	LOCAL CONST Robtarget Tr_meulage_bavure_P136 :=[[-151.101640625,13.911193359375,23],[0.363113173339064,-0.403939689053268,0.624425765586211,-0.561314541257626],[0,0,0,0],[8.999999E+09,8.999999E+09,8.999999E+09,8.999999E+09,8.999999E+09,8.999999E+09]];
	LOCAL CONST Robtarget Tr_meulage_bavure_P137 :=[[-149.937296875,16.62026953125,23],[0.361366142392558,-0.400488127447699,0.625160151915924,-0.564090910547419],[0,0,0,0],[8.999999E+09,8.999999E+09,8.999999E+09,8.999999E+09,8.999999E+09,8.999999E+09]];
	LOCAL CONST Robtarget Tr_meulage_bavure_P138 :=[[-148.7885625,19.131255859375,23],[0.359765710075978,-0.397152746767946,0.625734149066699,-0.566828990331279],[0,0,0,0],[8.999999E+09,8.999999E+09,8.999999E+09,8.999999E+09,8.999999E+09,8.999999E+09]];
	LOCAL CONST Robtarget Tr_meulage_bavure_P139 :=[[-148.23471875,20.335998046875,23],[0.358570112588793,-0.394222003460565,0.625973297444358,-0.569362729050853],[0,0,0,0],[8.999999E+09,8.999999E+09,8.999999E+09,8.999999E+09,8.999999E+09,8.999999E+09]];
	LOCAL CONST Robtarget Tr_meulage_bavure_P140 :=[[-145.765296875,25.489470703125,23],[0.35796569299165,-0.39191876694484,0.625767359146769,-0.571555294773763],[0,0,0,0],[8.999999E+09,8.999999E+09,8.999999E+09,8.999999E+09,8.999999E+09,8.999999E+09]];
	LOCAL CONST Robtarget Tr_meulage_bavure_P141 :=[[-144.20271875,28.765869140625,23],[0.358018242776586,-0.390330323158982,0.625091784203007,-0.573345827562799],[0,0,0,0],[8.999999E+09,8.999999E+09,8.999999E+09,8.999999E+09,8.999999E+09,8.999999E+09]];
	LOCAL CONST Robtarget Tr_meulage_bavure_P142 :=[[-143.79815625,29.5517578125,23],[0.358645064931337,-0.3893852969019,0.624023000869993,-0.57475916899361],[0,0,0,0],[8.999999E+09,8.999999E+09,8.999999E+09,8.999999E+09,8.999999E+09,8.999999E+09]];
	LOCAL CONST Robtarget Tr_meulage_bavure_P143 :=[[-142.6278125,32.183806640625,23],[0.359633831929679,-0.388864753981572,0.622717813839782,-0.575908182238306],[0,0,0,0],[8.999999E+09,8.999999E+09,8.999999E+09,8.999999E+09,8.999999E+09,8.999999E+09]];
	LOCAL CONST Robtarget Tr_meulage_bavure_P144 :=[[-141.08978125,35.4830625,23],[0.360692368664617,-0.388472413246163,0.621385243175179,-0.576949372907133],[0,0,0,0],[8.999999E+09,8.999999E+09,8.999999E+09,8.999999E+09,8.999999E+09,8.999999E+09]];
	LOCAL CONST Robtarget Tr_meulage_bavure_P145 :=[[-140.90496875,35.88940625,23],[0.36152355469278,-0.387927178958205,0.620241455843297,-0.578025743095594],[0,0,0,0],[8.999999E+09,8.999999E+09,8.999999E+09,8.999999E+09,8.999999E+09,8.999999E+09]];
	LOCAL CONST Robtarget Tr_meulage_bavure_P146 :=[[-140.313296875,37.1786796875,23],[0.361932466131916,-0.387033912571134,0.619420641915412,-0.579247536765284],[0,0,0,0],[8.999999E+09,8.999999E+09,8.999999E+09,8.999999E+09,8.999999E+09,8.999999E+09]];
	LOCAL CONST Robtarget Tr_meulage_bavure_P147 :=[[-139.0531875,39.5576171875,23],[0.361853147250191,-0.385747951920083,0.618973239019357,-0.580631506889248],[0,0,0,0],[8.999999E+09,8.999999E+09,8.999999E+09,8.999999E+09,8.999999E+09,8.999999E+09]];
	LOCAL CONST Robtarget Tr_meulage_bavure_P148 :=[[-138.05065625,41.53494140625,23],[0.361341124651924,-0.384146531890856,0.618865172241677,-0.582125357854981],[0,0,0,0],[8.999999E+09,8.999999E+09,8.999999E+09,8.999999E+09,8.999999E+09,8.999999E+09]];
	LOCAL CONST Robtarget Tr_meulage_bavure_P149 :=[[-136.388,44.438078125,23],[0.360507751556033,-0.382372963113046,0.619030246412353,-0.583632274788522],[0,0,0,0],[8.999999E+09,8.999999E+09,8.999999E+09,8.999999E+09,8.999999E+09,8.999999E+09]];
	LOCAL CONST Robtarget Tr_meulage_bavure_P150 :=[[-135.13509375,47.07137890625,23],[0.359446609197695,-0.380538333002904,0.619411292399243,-0.585079792079636],[0,0,0,0],[8.999999E+09,8.999999E+09,8.999999E+09,8.999999E+09,8.999999E+09,8.999999E+09]];
	LOCAL CONST Robtarget Tr_meulage_bavure_P151 :=[[-133.055,51.51773046875,23],[0.358189967630797,-0.378660333676248,0.61998050741984,-0.586464380170082],[0,0,0,0],[8.999999E+09,8.999999E+09,8.999999E+09,8.999999E+09,8.999999E+09,8.999999E+09]];
	LOCAL CONST Robtarget Tr_meulage_bavure_P152 :=[[-132.991484375,51.62383984375,23],[0.356688173346148,-0.376690925174669,0.620772461958371,-0.587808680065362],[0,0,0,0],[8.999999E+09,8.999999E+09,8.999999E+09,8.999999E+09,8.999999E+09,8.999999E+09]];
	LOCAL CONST Robtarget Tr_meulage_bavure_P153 :=[[-132.88184375,51.8467109375,23],[0.354871689037836,-0.374562381729461,0.621834258118938,-0.589144517026389],[0,0,0,0],[8.999999E+09,8.999999E+09,8.999999E+09,8.999999E+09,8.999999E+09,8.999999E+09]];
	LOCAL CONST Robtarget Tr_meulage_bavure_P154 :=[[-132.33325,52.87548828125,23],[0.352738855187171,-0.372246378330528,0.623153787667112,-0.590497494302203],[0,0,0,0],[8.999999E+09,8.999999E+09,8.999999E+09,8.999999E+09,8.999999E+09,8.999999E+09]];
	LOCAL CONST Robtarget Tr_meulage_bavure_P155 :=[[-129.2417578125,58.37216015625,23],[0.350372889166439,-0.36982520954016,0.624675359558615,-0.591818255958748],[0,0,0,0],[8.999999E+09,8.999999E+09,8.999999E+09,8.999999E+09,8.999999E+09,8.999999E+09]];
	LOCAL CONST Robtarget Tr_meulage_bavure_P156 :=[[-128.5902734375,59.6175234375,23],[0.347952755656077,-0.367462162625027,0.626275780687696,-0.593025366569001],[0,0,0,0],[8.999999E+09,8.999999E+09,8.999999E+09,8.999999E+09,8.999999E+09,8.999999E+09]];
	LOCAL CONST Robtarget Tr_meulage_bavure_P157 :=[[-128.01315625,60.49066015625,23],[0.345666878551163,-0.365345597032472,0.627836321567684,-0.594018987173004],[0,0,0,0],[8.999999E+09,8.999999E+09,8.999999E+09,8.999999E+09,8.999999E+09,8.999999E+09]];
	LOCAL CONST Robtarget Tr_meulage_bavure_P158 :=[[-126.7691640625,62.76187109375,23],[0.343644652538738,-0.363593971431505,0.629272863290692,-0.594746534454914],[0,0,0,0],[8.999999E+09,8.999999E+09,8.999999E+09,8.999999E+09,8.999999E+09,8.999999E+09]];
	LOCAL CONST Robtarget Tr_meulage_bavure_P159 :=[[-125.6860078125,64.59457421875,23],[0.341903861092431,-0.362214737571814,0.630573008552044,-0.595214175353287],[0,0,0,0],[8.999999E+09,8.999999E+09,8.999999E+09,8.999999E+09,8.999999E+09,8.999999E+09]];
	LOCAL CONST Robtarget Tr_meulage_bavure_P160 :=[[-124.4326484375,66.62625,23],[0.340355790714089,-0.361121197706101,0.63179741148611,-0.595467419036633],[0,0,0,0],[8.999999E+09,8.999999E+09,8.999999E+09,8.999999E+09,8.999999E+09,8.999999E+09]];
	LOCAL CONST Robtarget Tr_meulage_bavure_P161 :=[[-123.00375,69.2471953125,23],[0.338884891304971,-0.360167100503058,0.633005414582959,-0.59560123847176],[0,0,0,0],[8.999999E+09,8.999999E+09,8.999999E+09,8.999999E+09,8.999999E+09,8.999999E+09]];
	LOCAL CONST Robtarget Tr_meulage_bavure_P162 :=[[-122.3022734375,70.33459375,23],[0.33739329406918,-0.359234517684621,0.634249603211876,-0.595687642348424],[0,0,0,0],[8.999999E+09,8.999999E+09,8.999999E+09,8.999999E+09,8.999999E+09,8.999999E+09]];
	LOCAL CONST Robtarget Tr_meulage_bavure_P163 :=[[-121.89965625,71.103359375,23],[0.335824905230539,-0.358297647661144,0.635582135777234,-0.595717867272956],[0,0,0,0],[8.999999E+09,8.999999E+09,8.999999E+09,8.999999E+09,8.999999E+09,8.999999E+09]];
	LOCAL CONST Robtarget Tr_meulage_bavure_P164 :=[[-121.4621875,71.8283046875,23],[0.334205475423421,-0.35736441895173,0.636977751618542,-0.595698511167591],[0,0,0,0],[8.999999E+09,8.999999E+09,8.999999E+09,8.999999E+09,8.999999E+09,8.999999E+09]];
	LOCAL CONST Robtarget Tr_meulage_bavure_P165 :=[[-116.748078125,79.6233828125,23],[0.332558951177178,-0.356471847846565,0.638428689604975,-0.595601522810398],[0,0,0,0],[8.999999E+09,8.999999E+09,8.999999E+09,8.999999E+09,8.999999E+09,8.999999E+09]];
	LOCAL CONST Robtarget Tr_meulage_bavure_P166 :=[[-116.44934375,80.07165625,23],[0.33089213683516,-0.355635671324102,0.639935992215293,-0.595412116882034],[0,0,0,0],[8.999999E+09,8.999999E+09,8.999999E+09,8.999999E+09,8.999999E+09,8.999999E+09]];
	LOCAL CONST Robtarget Tr_meulage_bavure_P167 :=[[-115.361484375,81.8792109375,23],[0.329186352606248,-0.354835404169223,0.641511190202099,-0.595139961732823],[0,0,0,0],[8.999999E+09,8.999999E+09,8.999999E+09,8.999999E+09,8.999999E+09,8.999999E+09]];
	LOCAL CONST Robtarget Tr_meulage_bavure_P168 :=[[-112.9508046875,85.6936953125,23],[0.32739769262739,-0.354043304067062,0.64319165616197,-0.594784484625449],[0,0,0,0],[8.999999E+09,8.999999E+09,8.999999E+09,8.999999E+09,8.999999E+09,8.999999E+09]];
	LOCAL CONST Robtarget Tr_meulage_bavure_P169 :=[[-110.774625,89.2081015625,23],[0.325512172612704,-0.353248750896646,0.644988949272338,-0.59434535481274],[0,0,0,0],[8.999999E+09,8.999999E+09,8.999999E+09,8.999999E+09,8.999999E+09,8.999999E+09]];
	LOCAL CONST Robtarget Tr_meulage_bavure_P170 :=[[-110.4715,89.681578125,23],[0.323541727027112,-0.352470758041441,0.646900127086222,-0.593805810997026],[0,0,0,0],[8.999999E+09,8.999999E+09,8.999999E+09,8.999999E+09,8.999999E+09,8.999999E+09]];
	LOCAL CONST Robtarget Tr_meulage_bavure_P171 :=[[-110.3179609375,89.93865625,23],[0.321490986582534,-0.351726089874816,0.648929676846336,-0.593146337555642],[0,0,0,0],[8.999999E+09,8.999999E+09,8.999999E+09,8.999999E+09,8.999999E+09,8.999999E+09]];
	LOCAL CONST Robtarget Tr_meulage_bavure_P172 :=[[-108.4508984375,92.7417578125,23],[0.319339852371983,-0.350964788325318,0.6510751687394,-0.592407714917494],[0,0,0,0],[8.999999E+09,8.999999E+09,8.999999E+09,8.999999E+09,8.999999E+09,8.999999E+09]];
	LOCAL CONST Robtarget Tr_meulage_bavure_P173 :=[[-107.08996875,94.77328125,23],[0.316996000347298,-0.350097784864441,0.653399226164253,-0.59162025662141],[0,0,0,0],[8.999999E+09,8.999999E+09,8.999999E+09,8.999999E+09,8.999999E+09,8.999999E+09]];
	LOCAL CONST Robtarget Tr_meulage_bavure_P174 :=[[-105.537234375,96.8504296875,23],[0.314366480436105,-0.349013203905433,0.655953733645348,-0.590836863097259],[0,0,0,0],[8.999999E+09,8.999999E+09,8.999999E+09,8.999999E+09,8.999999E+09,8.999999E+09]];
	LOCAL CONST Robtarget Tr_meulage_bavure_P175 :=[[-104.5172421875,98.662203125,23],[0.311427948746812,-0.347654360016432,0.658738048574652,-0.590095976991012],[0,0,0,0],[8.999999E+09,8.999999E+09,8.999999E+09,8.999999E+09,8.999999E+09,8.999999E+09]];
	LOCAL CONST Robtarget Tr_meulage_bavure_P176 :=[[-104.1592421875,99.2328828125,23],[0.308276601042876,-0.346110430708768,0.661687715989301,-0.589357678759601],[0,0,0,0],[8.999999E+09,8.999999E+09,8.999999E+09,8.999999E+09,8.999999E+09,8.999999E+09]];
	LOCAL CONST Robtarget Tr_meulage_bavure_P177 :=[[-103.0036953125,100.7189609375,23],[0.305135247230992,-0.344604748309039,0.664658435505481,-0.588531403114186],[0,0,0,0],[8.999999E+09,8.999999E+09,8.999999E+09,8.999999E+09,8.999999E+09,8.999999E+09]];
	LOCAL CONST Robtarget Tr_meulage_bavure_P178 :=[[-102.00121875,102.1814609375,23],[0.302287241198627,-0.343432763280974,0.66747032690831,-0.587502956256929],[0,0,0,0],[8.999999E+09,8.999999E+09,8.999999E+09,8.999999E+09,8.999999E+09,8.999999E+09]];
	LOCAL CONST Robtarget Tr_meulage_bavure_P179 :=[[-97.7013515625,108.074984375,23],[0.299987070179315,-0.342864199056344,0.669960522310556,-0.586178127599494],[0,0,0,0],[8.999999E+09,8.999999E+09,8.999999E+09,8.999999E+09,8.999999E+09,8.999999E+09]];
	LOCAL CONST Robtarget Tr_meulage_bavure_P180 :=[[-97.20065625,108.7268046875,23],[0.298390218171339,-0.343046324630686,0.672013629572218,-0.584534155140837],[0,0,0,0],[8.999999E+09,8.999999E+09,8.999999E+09,8.999999E+09,8.999999E+09,8.999999E+09]];
	LOCAL CONST Robtarget Tr_meulage_bavure_P181 :=[[-96.925140625,109.1156953125,23],[0.297488777694042,-0.343974793916163,0.673625579809489,-0.582589346386258],[0,0,0,0],[8.999999E+09,8.999999E+09,8.999999E+09,8.999999E+09,8.999999E+09,8.999999E+09]];
	LOCAL CONST Robtarget Tr_meulage_bavure_P182 :=[[-96.654234375,109.4932890625,23],[0.297146717753407,-0.345460993457581,0.674847244361684,-0.58046681809137],[0,0,0,0],[8.999999E+09,8.999999E+09,8.999999E+09,8.999999E+09,8.999999E+09,8.999999E+09]];
	LOCAL CONST Robtarget Tr_meulage_bavure_P183 :=[[-93.7308671875,113.3792734375,23],[0.297098761957459,-0.347164074281642,0.675810702966835,-0.578350520815005],[0,0,0,0],[8.999999E+09,8.999999E+09,8.999999E+09,8.999999E+09,8.999999E+09,8.999999E+09]];
	LOCAL CONST Robtarget Tr_meulage_bavure_P184 :=[[-90.1459375,118.35940625,23],[0.296995083840805,-0.348662276006968,0.6767185983147,-0.576437746993568],[0,0,0,0],[8.999999E+09,8.999999E+09,8.999999E+09,8.999999E+09,8.999999E+09,8.999999E+09]];
	LOCAL CONST Robtarget Tr_meulage_bavure_P185 :=[[-89.706484375,118.935421875,23],[0.296477938104876,-0.34949723785255,0.677774921241467,-0.574955362690569],[0,0,0,0],[8.999999E+09,8.999999E+09,8.999999E+09,8.999999E+09,8.999999E+09,8.999999E+09]];
	LOCAL CONST Robtarget Tr_meulage_bavure_P186 :=[[-89.5105,119.176546875,23],[0.295232063451212,-0.349274248056214,0.679170511051546,-0.574084440890961],[0,0,0,0],[8.999999E+09,8.999999E+09,8.999999E+09,8.999999E+09,8.999999E+09,8.999999E+09]];
	LOCAL CONST Robtarget Tr_meulage_bavure_P187 :=[[-89.0611875,119.83196875,23],[0.293080552541801,-0.347759738084034,0.681007104196331,-0.573930551829787],[0,0,0,0],[8.999999E+09,8.999999E+09,8.999999E+09,8.999999E+09,8.999999E+09,8.999999E+09]];
	LOCAL CONST Robtarget Tr_meulage_bavure_P188 :=[[-87.366484375,122.046390625,23],[0.290040566264844,-0.344934373310814,0.683249092361541,-0.574514948296887],[0,0,0,0],[8.999999E+09,8.999999E+09,8.999999E+09,8.999999E+09,8.999999E+09,8.999999E+09]];
	LOCAL CONST Robtarget Tr_meulage_bavure_P189 :=[[-85.4241328125,124.5614921875,23],[0.286302590251918,-0.341056323606131,0.685782309095291,-0.575685708937823],[0,0,0,0],[8.999999E+09,8.999999E+09,8.999999E+09,8.999999E+09,8.999999E+09,8.999999E+09]];
	LOCAL CONST Robtarget Tr_meulage_bavure_P190 :=[[-82.9652109375,127.53896875,23],[0.282238780633603,-0.336559090185623,0.688360590316553,-0.577259861084182],[0,0,0,0],[8.999999E+09,8.999999E+09,8.999999E+09,8.999999E+09,8.999999E+09,8.999999E+09]];
	LOCAL CONST Robtarget Tr_meulage_bavure_P191 :=[[-80.8466171875,130.312015625,23],[0.278274994959359,-0.331954569840343,0.690722014669287,-0.579027019398648],[0,0,0,0],[8.999999E+09,8.999999E+09,8.999999E+09,8.999999E+09,8.999999E+09,8.999999E+09]];
	LOCAL CONST Robtarget Tr_meulage_bavure_P192 :=[[-80.806546875,130.3608671875,23],[0.274742616549122,-0.327682985270072,0.692696966908732,-0.580785044445601],[0,0,0,0],[8.999999E+09,8.999999E+09,8.999999E+09,8.999999E+09,8.999999E+09,8.999999E+09]];
	LOCAL CONST Robtarget Tr_meulage_bavure_P193 :=[[-80.775234375,130.400515625,23],[0.271819685652551,-0.323980055433208,0.694203028496095,-0.582437239022449],[0,0,0,0],[8.999999E+09,8.999999E+09,8.999999E+09,8.999999E+09,8.999999E+09,8.999999E+09]];
	LOCAL CONST Robtarget Tr_meulage_bavure_P194 :=[[-80.66,130.534453125,23],[0.269492995590509,-0.320855422562745,0.69527098544135,-0.583972242442352],[0,0,0,0],[8.999999E+09,8.999999E+09,8.999999E+09,8.999999E+09,8.999999E+09,8.999999E+09]];
	LOCAL CONST Robtarget Tr_meulage_bavure_P195 :=[[-75.0816015625,136.849671875,23],[0.267608889300657,-0.318155220259668,0.696010587349302,-0.585433173373759],[0,0,0,0],[8.999999E+09,8.999999E+09,8.999999E+09,8.999999E+09,8.999999E+09,8.999999E+09]];
	LOCAL CONST Robtarget Tr_meulage_bavure_P196 :=[[-73.9031640625,138.106265625,23],[0.265971457519477,-0.315679629512676,0.696553803832876,-0.586871667114418],[0,0,0,0],[8.999999E+09,8.999999E+09,8.999999E+09,8.999999E+09,8.999999E+09,8.999999E+09]];
	LOCAL CONST Robtarget Tr_meulage_bavure_P197 :=[[-70.499453125,142.30071875,23],[0.264424748051487,-0.313302265360263,0.697024796870706,-0.588283669402258],[0,0,0,0],[8.999999E+09,8.999999E+09,8.999999E+09,8.999999E+09,8.999999E+09,8.999999E+09]];
	LOCAL CONST Robtarget Tr_meulage_bavure_P198 :=[[-69.435421875,143.518640625,23],[0.262940352786829,-0.311003055889999,0.69744901940964,-0.589664595705009],[0,0,0,0],[8.999999E+09,8.999999E+09,8.999999E+09,8.999999E+09,8.999999E+09,8.999999E+09]];
	LOCAL CONST Robtarget Tr_meulage_bavure_P199 :=[[-67.65221875,145.57946875,23],[0.26158305272051,-0.308882913750533,0.697810610604228,-0.590953470123117],[0,0,0,0],[8.999999E+09,8.999999E+09,8.999999E+09,8.999999E+09,8.999999E+09,8.999999E+09]];
	LOCAL CONST Robtarget Tr_meulage_bavure_P200 :=[[-63.85848828125,149.82321875,23],[0.260452446063248,-0.307115703409703,0.698100327852684,-0.592030742707512],[0,0,0,0],[8.999999E+09,8.999999E+09,8.999999E+09,8.999999E+09,8.999999E+09,8.999999E+09]];
	LOCAL CONST Robtarget Tr_meulage_bavure_P201 :=[[-62.9795546875,150.73965625,23],[0.259650622045114,-0.305842532734676,0.698285923040029,-0.592822628891778],[0,0,0,0],[8.999999E+09,8.999999E+09,8.999999E+09,8.999999E+09,8.999999E+09,8.999999E+09]];
	LOCAL CONST Robtarget Tr_meulage_bavure_P202 :=[[-60.04244921875,154.120734375,23],[0.25923435549752,-0.305149200328328,0.698357387354537,-0.593277737654222],[0,0,0,0],[8.999999E+09,8.999999E+09,8.999999E+09,8.999999E+09,8.999999E+09,8.999999E+09]];
	LOCAL CONST Robtarget Tr_meulage_bavure_P203 :=[[-58.3733515625,155.91925,23],[0.259193420326712,-0.305039549462365,0.698335046608728,-0.593378299907507],[0,0,0,0],[8.999999E+09,8.999999E+09,8.999999E+09,8.999999E+09,8.999999E+09,8.999999E+09]];
	LOCAL CONST Robtarget Tr_meulage_bavure_P204 :=[[-57.8063046875,156.5224375,23],[0.259457229635472,-0.305442867370749,0.698264748264398,-0.593138215000077],[0,0,0,0],[8.999999E+09,8.999999E+09,8.999999E+09,8.999999E+09,8.999999E+09,8.999999E+09]];
	LOCAL CONST Robtarget Tr_meulage_bavure_P205 :=[[-53.8414921875,160.451046875,23],[0.259910866387483,-0.306232150271341,0.698209736878708,-0.592597143936473],[0,0,0,0],[8.999999E+09,8.999999E+09,8.999999E+09,8.999999E+09,8.999999E+09,8.999999E+09]];
	LOCAL CONST Robtarget Tr_meulage_bavure_P206 :=[[-51.208921875,163.25109375,23],[0.260395135511095,-0.307211321910998,0.698243437299184,-0.591837544737132],[0,0,0,0],[8.999999E+09,8.999999E+09,8.999999E+09,8.999999E+09,8.999999E+09,8.999999E+09]];
	LOCAL CONST Robtarget Tr_meulage_bavure_P207 :=[[-48.69293359375,165.973234375,23],[0.260708052450437,-0.308133124993847,0.698462495975598,-0.590961445768304],[0,0,0,0],[8.999999E+09,8.999999E+09,8.999999E+09,8.999999E+09,8.999999E+09,8.999999E+09]];
	LOCAL CONST Robtarget Tr_meulage_bavure_P208 :=[[-47.96395703125,166.6900625,23],[0.260627562818114,-0.308725558365438,0.698976562907696,-0.590079289263047],[0,0,0,0],[8.999999E+09,8.999999E+09,8.999999E+09,8.999999E+09,8.999999E+09,8.999999E+09]];
	LOCAL CONST Robtarget Tr_meulage_bavure_P209 :=[[-47.6884453125,166.9998125,23],[0.259952138246991,-0.308717659214279,0.699872182769465,-0.589319285697981],[0,0,0,0],[8.999999E+09,8.999999E+09,8.999999E+09,8.999999E+09,8.999999E+09,8.999999E+09]];
	LOCAL CONST Robtarget Tr_meulage_bavure_P210 :=[[-47.49398828125,167.2056875,23],[0.258524685420064,-0.307880894401815,0.70120753717733,-0.588797360470051],[0,0,0,0],[8.999999E+09,8.999999E+09,8.999999E+09,8.999999E+09,8.999999E+09,8.999999E+09]];
	LOCAL CONST Robtarget Tr_meulage_bavure_P211 :=[[-46.68640234375,168.037875,23],[0.256255031366667,-0.306077422500699,0.703012135818707,-0.588577868447512],[0,0,0,0],[8.999999E+09,8.999999E+09,8.999999E+09,8.999999E+09,8.999999E+09,8.999999E+09]];
	LOCAL CONST Robtarget Tr_meulage_bavure_P212 :=[[-42.5556953125,172.1044375,23],[0.253174527212128,-0.303299309659537,0.705237754876775,-0.588686586077285],[0,0,0,0],[8.999999E+09,8.999999E+09,8.999999E+09,8.999999E+09,8.999999E+09,8.999999E+09]];
	LOCAL CONST Robtarget Tr_meulage_bavure_P213 :=[[-41.41424609375,173.362859375,23],[0.249437788419242,-0.299696304442926,0.707774725152081,-0.589082212639006],[0,0,0,0],[8.999999E+09,8.999999E+09,8.999999E+09,8.999999E+09,8.999999E+09,8.999999E+09]];
	LOCAL CONST Robtarget Tr_meulage_bavure_P214 :=[[-39.20593359375,175.651515625,23],[0.245328958803579,-0.29556827111994,0.710440992387538,-0.589683555320082],[0,0,0,0],[8.999999E+09,8.999999E+09,8.999999E+09,8.999999E+09,8.999999E+09,8.999999E+09]];
	LOCAL CONST Robtarget Tr_meulage_bavure_P215 :=[[-34.94815234375,180.011390625,23],[0.241200692788689,-0.291315873340678,0.713035034890375,-0.590371346490408],[0,0,0,0],[8.999999E+09,8.999999E+09,8.999999E+09,8.999999E+09,8.999999E+09,8.999999E+09]];
	LOCAL CONST Robtarget Tr_meulage_bavure_P216 :=[[-34.57086328125,180.35953125,23],[0.237386947714952,-0.287326399661774,0.71537675117121,-0.591038984328196],[0,0,0,0],[8.999999E+09,8.999999E+09,8.999999E+09,8.999999E+09,8.999999E+09,8.999999E+09]];
	LOCAL CONST Robtarget Tr_meulage_bavure_P217 :=[[-33.607484375,181.285671875,23],[0.234098705180864,-0.283854988465174,0.717364032824637,-0.591618953521312],[0,0,0,0],[8.999999E+09,8.999999E+09,8.999999E+09,8.999999E+09,8.999999E+09,8.999999E+09]];
	LOCAL CONST Robtarget Tr_meulage_bavure_P218 :=[[-32.24230859375,182.4925,23],[0.231389418192959,-0.28095490120141,0.718964421329079,-0.592126204032698],[0,0,0,0],[8.999999E+09,8.999999E+09,8.999999E+09,8.999999E+09,8.999999E+09,8.999999E+09]];
	LOCAL CONST Robtarget Tr_meulage_bavure_P219 :=[[-31.390533203125,183.272,23],[0.229147339722196,-0.27850899502818,0.720247483284206,-0.592594126877242],[0,0,0,0],[8.999999E+09,8.999999E+09,8.999999E+09,8.999999E+09,8.999999E+09,8.999999E+09]];
	LOCAL CONST Robtarget Tr_meulage_bavure_P220 :=[[-26.916779296875,187.099859375,23],[0.227187311028143,-0.276294003133417,0.721302168803879,-0.593102630932568],[0,0,0,0],[8.999999E+09,8.999999E+09,8.999999E+09,8.999999E+09,8.999999E+09,8.999999E+09]];
	LOCAL CONST Robtarget Tr_meulage_bavure_P221 :=[[-24.466033203125,189.348875,23],[0.225315180737453,-0.274084145121572,0.722226163804524,-0.593717373030659],[0,0,0,0],[8.999999E+09,8.999999E+09,8.999999E+09,8.999999E+09,8.999999E+09,8.999999E+09]];
	LOCAL CONST Robtarget Tr_meulage_bavure_P222 :=[[-20.982390625,192.370671875,23],[0.223403102383008,-0.271738206161415,0.723087604344703,-0.594469273891311],[0,0,0,0],[8.999999E+09,8.999999E+09,8.999999E+09,8.999999E+09,8.999999E+09,8.999999E+09]];
	LOCAL CONST Robtarget Tr_meulage_bavure_P223 :=[[-19.10336328125,194.2511875,23],[0.221425398857496,-0.269241274270312,0.723908292677629,-0.595345876581553],[0,0,0,0],[8.999999E+09,8.999999E+09,8.999999E+09,8.999999E+09,8.999999E+09,8.999999E+09]];
	LOCAL CONST Robtarget Tr_meulage_bavure_P224 :=[[-18.80859375,194.504453125,23],[0.21942139915103,-0.266659496341684,0.724682721879693,-0.596306896836221],[0,0,0,0],[8.999999E+09,8.999999E+09,8.999999E+09,8.999999E+09,8.999999E+09,8.999999E+09]];
	LOCAL CONST Robtarget Tr_meulage_bavure_P225 :=[[-15.535796875,197.271734375,23],[0.217482339471062,-0.264111761664924,0.725374934386033,-0.597308642104651],[0,0,0,0],[8.999999E+09,8.999999E+09,8.999999E+09,8.999999E+09,8.999999E+09,8.999999E+09]];
	LOCAL CONST Robtarget Tr_meulage_bavure_P226 :=[[-14.38656640625,198.22653125,23],[0.215685475116499,-0.261691661864608,0.725950038924085,-0.598325823377556],[0,0,0,0],[8.999999E+09,8.999999E+09,8.999999E+09,8.999999E+09,8.999999E+09,8.999999E+09]];
	LOCAL CONST Robtarget Tr_meulage_bavure_P227 :=[[-14.2441708984375,198.341984375,23],[0.214071327561037,-0.259461487748869,0.726403020672261,-0.59932616716577],[0,0,0,0],[8.999999E+09,8.999999E+09,8.999999E+09,8.999999E+09,8.999999E+09,8.999999E+09]];
	LOCAL CONST Robtarget Tr_meulage_bavure_P228 :=[[-13.9234921875,198.62090625,23],[0.212656773606905,-0.257433136373764,0.726720308684264,-0.600318973448047],[0,0,0,0],[8.999999E+09,8.999999E+09,8.999999E+09,8.999999E+09,8.999999E+09,8.999999E+09]];
	LOCAL CONST Robtarget Tr_meulage_bavure_P229 :=[[-6.44500732421875,204.744109375,23],[0.211343507043338,-0.255486294409757,0.726943875156387,-0.60134289533677],[0,0,0,0],[8.999999E+09,8.999999E+09,8.999999E+09,8.999999E+09,8.999999E+09,8.999999E+09]];
	LOCAL CONST Robtarget Tr_meulage_bavure_P230 :=[[-4.770416015625,206.066828125,23],[0.209903474101674,-0.253333301261567,0.727157715519496,-0.602498486962774],[0,0,0,0],[8.999999E+09,8.999999E+09,8.999999E+09,8.999999E+09,8.999999E+09,8.999999E+09]];
	LOCAL CONST Robtarget Tr_meulage_bavure_P231 :=[[-1.2413330078125,208.911890625,23],[0.207823352269298,-0.25031838984503,0.727533303346977,-0.604024379042748],[0,0,0,0],[8.999999E+09,8.999999E+09,8.999999E+09,8.999999E+09,8.999999E+09,8.999999E+09]];
	LOCAL CONST Robtarget Tr_meulage_bavure_P232 :=[[1.50991821289063,211.015375,23],[0.204213513188322,-0.245379488056485,0.728416370025912,-0.606213938928076],[0,0,0,0],[8.999999E+09,8.999999E+09,8.999999E+09,8.999999E+09,8.999999E+09,8.999999E+09]];
	LOCAL CONST Robtarget Tr_meulage_bavure_P233 :=[[5.3576357421875,214.052484375,23],[0.197930878967157,-0.237150606750637,0.730189298230088,-0.609431329699536],[0,0,0,0],[8.999999E+09,8.999999E+09,8.999999E+09,8.999999E+09,8.999999E+09,8.999999E+09]];
	LOCAL CONST Robtarget Tr_meulage_bavure_P234 :=[[6.84130859375,215.1638125,23],[0.187712989087851,-0.224125457327204,0.733141487562592,-0.614031898454865],[0,0,0,0],[8.999999E+09,8.999999E+09,8.999999E+09,8.999999E+09,8.999999E+09,8.999999E+09]];
	LOCAL CONST Robtarget Tr_meulage_bavure_P235 :=[[7.3984072265625,215.63,23],[0.172504478983547,-0.20511598853545,0.737325338971367,-0.620097557234745],[0,0,0,0],[8.999999E+09,8.999999E+09,8.999999E+09,8.999999E+09,8.999999E+09,8.999999E+09]];
	LOCAL CONST Robtarget Tr_meulage_bavure_P236 :=[[9.3818056640625,217.564265625,23],[0.151549893185851,-0.17931796598194,0.74241703056212,-0.627450914162041],[0,0,0,0],[8.999999E+09,8.999999E+09,8.999999E+09,8.999999E+09,8.999999E+09,8.999999E+09]];
	LOCAL CONST Robtarget Tr_meulage_bavure_P237 :=[[11.914978515625,219.3876875,23],[0.124220420395778,-0.146146884846895,0.747803441259262,-0.635610248853061],[0,0,0,0],[8.999999E+09,8.999999E+09,8.999999E+09,8.999999E+09,8.999999E+09,8.999999E+09]];
	LOCAL CONST Robtarget Tr_meulage_bavure_P238 :=[[12.1049501953125,219.532171875,23],[0.0897657639649963,-0.104927499133286,0.752592704605305,-0.643845127744466],[0,0,0,0],[8.999999E+09,8.999999E+09,8.999999E+09,8.999999E+09,8.999999E+09,8.999999E+09]];
	LOCAL CONST Robtarget Tr_meulage_bavure_P239 :=[[14.768951171875,220.201109375,23],[0.0471999623288128,-0.0547682552860186,0.755523575206771,-0.651119596599475],[0,0,0,0],[8.999999E+09,8.999999E+09,8.999999E+09,8.999999E+09,8.999999E+09,8.999999E+09]];
	LOCAL CONST Robtarget Tr_meulage_bavure_P240 :=[[15.1896669921875,220.290953125,23],[0.00391673808409907,-0.00450800521522732,-0.754862835226616,0.655855500125901],[0,0,0,0],[8.999999E+09,8.999999E+09,8.999999E+09,8.999999E+09,8.999999E+09,8.999999E+09]];
	LOCAL CONST Robtarget Tr_meulage_bavure_P241 :=[[15.542328125,220.304265625,23],[0.0619053642117967,-0.0706232456407094,-0.748672202083587,0.656254536658063],[0,0,0,0],[8.999999E+09,8.999999E+09,8.999999E+09,8.999999E+09,8.999999E+09,8.999999E+09]];
	LOCAL CONST Robtarget Tr_meulage_bavure_P242 :=[[17.782501953125,220.00159375,23],[0.121896077477367,-0.137740018820242,-0.736087584245498,0.651416995349874],[0,0,0,0],[8.999999E+09,8.999999E+09,8.999999E+09,8.999999E+09,8.999999E+09,8.999999E+09]];
	LOCAL CONST Robtarget Tr_meulage_bavure_P243 :=[[19.011505859375,219.1355625,23],[0.177301752020205,-0.198335874044401,-0.718667958085683,0.642451037681912],[0,0,0,0],[8.999999E+09,8.999999E+09,8.999999E+09,8.999999E+09,8.999999E+09,8.999999E+09]];
	LOCAL CONST Robtarget Tr_meulage_bavure_P244 :=[[20.29995703125,218.304328125,23],[0.223287940782648,-0.247145069123424,-0.699644445371508,0.632107158929416],[0,0,0,0],[8.999999E+09,8.999999E+09,8.999999E+09,8.999999E+09,8.999999E+09,8.999999E+09]];
	LOCAL CONST Robtarget Tr_meulage_bavure_P245 :=[[22.17059375,216.388125,23],[0.258324297897703,-0.282817710648907,-0.682044025541808,0.622975639075634],[0,0,0,0],[8.999999E+09,8.999999E+09,8.999999E+09,8.999999E+09,8.999999E+09,8.999999E+09]];
	LOCAL CONST Robtarget Tr_meulage_bavure_P246 :=[[22.943115234375,215.523125,23],[0.283277734737214,-0.306695210666897,-0.667508852587879,0.616541729709315],[0,0,0,0],[8.999999E+09,8.999999E+09,8.999999E+09,8.999999E+09,8.999999E+09,8.999999E+09]];
	LOCAL CONST Robtarget Tr_meulage_bavure_P247 :=[[23.142974609375,215.210390625,23],[0.300023695928356,-0.321167914354036,-0.656391604412083,0.613177799931064],[0,0,0,0],[8.999999E+09,8.999999E+09,8.999999E+09,8.999999E+09,8.999999E+09,8.999999E+09]];
	LOCAL CONST Robtarget Tr_meulage_bavure_P248 :=[[26.006591796875,211.0040625,23],[0.310535323951501,-0.328675620854283,-0.648327618742999,0.612545057615699],[0,0,0,0],[8.999999E+09,8.999999E+09,8.999999E+09,8.999999E+09,8.999999E+09,8.999999E+09]];
	LOCAL CONST Robtarget Tr_meulage_bavure_P249 :=[[28.899353515625,206.60128125,23],[0.316651094086674,-0.331390976815339,-0.642583469500546,0.614002108973355],[0,0,0,0],[8.999999E+09,8.999999E+09,8.999999E+09,8.999999E+09,8.999999E+09,8.999999E+09]];
	LOCAL CONST Robtarget Tr_meulage_bavure_P250 :=[[29.728302734375,205.386140625,23],[0.319945859614084,-0.331125911864109,-0.638374760442697,0.616820835119645],[0,0,0,0],[8.999999E+09,8.999999E+09,8.999999E+09,8.999999E+09,8.999999E+09,8.999999E+09]];
	LOCAL CONST Robtarget Tr_meulage_bavure_P251 :=[[30.96243359375,203.584171875,23],[0.321654675156927,-0.329279286634659,-0.635048726900972,0.620343885118985],[0,0,0,0],[8.999999E+09,8.999999E+09,8.999999E+09,8.999999E+09,8.999999E+09,8.999999E+09]];
	LOCAL CONST Robtarget Tr_meulage_bavure_P252 :=[[33.2144453125,200.487359375,23],[0.322686819263229,-0.32682954352752,-0.632107868709676,0.624095592410877],[0,0,0,0],[8.999999E+09,8.999999E+09,8.999999E+09,8.999999E+09,8.999999E+09,8.999999E+09]];
	LOCAL CONST Robtarget Tr_meulage_bavure_P253 :=[[37.9583125,194.060453125,23],[0.32350539086071,-0.324284803632072,-0.629319117331403,0.627806559999648],[0,0,0,0],[8.999999E+09,8.999999E+09,8.999999E+09,8.999999E+09,8.999999E+09,8.999999E+09]];
	LOCAL CONST Robtarget Tr_meulage_bavure_P254 :=[[40.1090703125,190.888578125,23],[0.324290887764197,-0.321831108466618,-0.626592214962344,0.631381306252284],[0,0,0,0],[8.999999E+09,8.999999E+09,8.999999E+09,8.999999E+09,8.999999E+09,8.999999E+09]];
	LOCAL CONST Robtarget Tr_meulage_bavure_P255 :=[[41.9234609375,188.34921875,23],[0.325084104557967,-0.319520541726406,-0.623920104777116,0.634783940592011],[0,0,0,0],[8.999999E+09,8.999999E+09,8.999999E+09,8.999999E+09,8.999999E+09,8.999999E+09]];
	LOCAL CONST Robtarget Tr_meulage_bavure_P256 :=[[44.363984375,184.8478125,23],[0.325855209154127,-0.317341781965301,-0.621337589605405,0.638006407357757],[0,0,0,0],[8.999999E+09,8.999999E+09,8.999999E+09,8.999999E+09,8.999999E+09,8.999999E+09]];
	LOCAL CONST Robtarget Tr_meulage_bavure_P257 :=[[45.731140625,182.934078125,23],[0.326647599437521,-0.31532852810653,-0.618822907630602,0.641036250250703],[0,0,0,0],[8.999999E+09,8.999999E+09,8.999999E+09,8.999999E+09,8.999999E+09,8.999999E+09]];
	LOCAL CONST Robtarget Tr_meulage_bavure_P258 :=[[47.5583515625,180.494078125,23],[0.327475417388791,-0.313503038011105,-0.616382739818725,0.643854031762951],[0,0,0,0],[8.999999E+09,8.999999E+09,8.999999E+09,8.999999E+09,8.999999E+09,8.999999E+09]];
	LOCAL CONST Robtarget Tr_meulage_bavure_P259 :=[[50.40579296875,176.811125,23],[0.328207818464939,-0.311757482224153,-0.614100318846837,0.646504213882598],[0,0,0,0],[8.999999E+09,8.999999E+09,8.999999E+09,8.999999E+09,8.999999E+09,8.999999E+09]];
	LOCAL CONST Robtarget Tr_meulage_bavure_P260 :=[[51.00183203125,175.88040625,23],[0.328573075772817,-0.309849251220576,-0.61211957416854,0.649109237582523],[0,0,0,0],[8.999999E+09,8.999999E+09,8.999999E+09,8.999999E+09,8.999999E+09,8.999999E+09]];
	LOCAL CONST Robtarget Tr_meulage_bavure_P261 :=[[54.5407734375,170.242578125,23],[0.328239021625795,-0.307486597313832,-0.610608761702741,0.651819052564703],[0,0,0,0],[8.999999E+09,8.999999E+09,8.999999E+09,8.999999E+09,8.999999E+09,8.999999E+09]];
	LOCAL CONST Robtarget Tr_meulage_bavure_P262 :=[[55.1708359375,169.26940625,23],[0.327088298193951,-0.304577764446545,-0.609623509202251,0.654679163878967],[0,0,0,0],[8.999999E+09,8.999999E+09,8.999999E+09,8.999999E+09,8.999999E+09,8.999999E+09]];
	LOCAL CONST Robtarget Tr_meulage_bavure_P263 :=[[55.540953125,168.720125,23],[0.325442042663654,-0.301449749292493,-0.609025614396537,0.657497776823103],[0,0,0,0],[8.999999E+09,8.999999E+09,8.999999E+09,8.999999E+09,8.999999E+09,8.999999E+09]];
	LOCAL CONST Robtarget Tr_meulage_bavure_P264 :=[[57.8688984375,165.123359375,23],[0.324070575547063,-0.298828874169683,-0.608477462969558,0.659874793491314],[0,0,0,0],[8.999999E+09,8.999999E+09,8.999999E+09,8.999999E+09,8.999999E+09,8.999999E+09]];
	LOCAL CONST Robtarget Tr_meulage_bavure_P265 :=[[58.964875,163.68078125,23],[0.323887940233861,-0.297551595101223,-0.60758493145613,0.661362382881908],[0,0,0,0],[8.999999E+09,8.999999E+09,8.999999E+09,8.999999E+09,8.999999E+09,8.999999E+09]];
	LOCAL CONST Robtarget Tr_meulage_bavure_P266 :=[[59.75341796875,162.826078125,23],[0.325471245652895,-0.298143385517853,-0.606112862492925,0.661669243539201],[0,0,0,0],[8.999999E+09,8.999999E+09,8.999999E+09,8.999999E+09,8.999999E+09,8.999999E+09]];
	LOCAL CONST Robtarget Tr_meulage_bavure_P267 :=[[60.56955078125,161.5953125,23],[0.328708240927848,-0.300493898546605,-0.604112523918591,0.660834599371955],[0,0,0,0],[8.999999E+09,8.999999E+09,8.999999E+09,8.999999E+09,8.999999E+09,8.999999E+09]];
	LOCAL CONST Robtarget Tr_meulage_bavure_P268 :=[[65.628234375,155.054875,23],[0.3327826342601,-0.303853641429328,-0.6019353952919,0.659243856869239],[0,0,0,0],[8.999999E+09,8.999999E+09,8.999999E+09,8.999999E+09,8.999999E+09,8.999999E+09]];
	LOCAL CONST Robtarget Tr_meulage_bavure_P269 :=[[66.6651953125,153.306671875,23],[0.336510464509657,-0.307144134428822,-0.600110733787954,0.657487866925274],[0,0,0,0],[8.999999E+09,8.999999E+09,8.999999E+09,8.999999E+09,8.999999E+09,8.999999E+09]];
	LOCAL CONST Robtarget Tr_meulage_bavure_P270 :=[[67.4820859375,152.073890625,23],[0.338883299771561,-0.309438452981514,-0.599102917366099,0.656111002312699],[0,0,0,0],[8.999999E+09,8.999999E+09,8.999999E+09,8.999999E+09,8.999999E+09,8.999999E+09]];
	LOCAL CONST Robtarget Tr_meulage_bavure_P271 :=[[68.479765625,150.469703125,23],[0.339450276856727,-0.310319109130537,-0.599131786020222,0.655375207824145],[0,0,0,0],[8.999999E+09,8.999999E+09,8.999999E+09,8.999999E+09,8.999999E+09,8.999999E+09]];
	LOCAL CONST Robtarget Tr_meulage_bavure_P272 :=[[70.648921875,147.182921875,23],[0.338393689015913,-0.30993009048273,-0.600103683194316,0.655216467790748],[0,0,0,0],[8.999999E+09,8.999999E+09,8.999999E+09,8.999999E+09,8.999999E+09,8.999999E+09]];
	LOCAL CONST Robtarget Tr_meulage_bavure_P273 :=[[72.7957734375,143.80371875,23],[0.336348123469612,-0.30882132431058,-0.601698361263421,0.65533076499005],[0,0,0,0],[8.999999E+09,8.999999E+09,8.999999E+09,8.999999E+09,8.999999E+09,8.999999E+09]];
	LOCAL CONST Robtarget Tr_meulage_bavure_P274 :=[[73.6694921875,142.54796875,23],[0.334055940460113,-0.307636637570664,-0.603537979314405,0.655368778164332],[0,0,0,0],[8.999999E+09,8.999999E+09,8.999999E+09,8.999999E+09,8.999999E+09,8.999999E+09]];
	LOCAL CONST Robtarget Tr_meulage_bavure_P275 :=[[77.3621484375,137.8243125,23],[0.332108727010819,-0.306894954950528,-0.605325432708239,0.655057555170346],[0,0,0,0],[8.999999E+09,8.999999E+09,8.999999E+09,8.999999E+09,8.999999E+09,8.999999E+09]];
	LOCAL CONST Robtarget Tr_meulage_bavure_P276 :=[[77.391140625,137.78259375,23],[0.330809905167146,-0.306849701794436,-0.606894564826024,0.654283619187123],[0,0,0,0],[8.999999E+09,8.999999E+09,8.999999E+09,8.999999E+09,8.999999E+09,8.999999E+09]];
	LOCAL CONST Robtarget Tr_meulage_bavure_P277 :=[[79.7291875,134.655296875,23],[0.330205811253363,-0.307517720793344,-0.608194982684563,0.653066487158773],[0,0,0,0],[8.999999E+09,8.999999E+09,8.999999E+09,8.999999E+09,8.999999E+09,8.999999E+09]];
	LOCAL CONST Robtarget Tr_meulage_bavure_P278 :=[[80.649140625,133.351984375,23],[0.330189821133415,-0.308785957025888,-0.60925498083289,0.651486210977489],[0,0,0,0],[8.999999E+09,8.999999E+09,8.999999E+09,8.999999E+09,8.999999E+09,8.999999E+09]];
	LOCAL CONST Robtarget Tr_meulage_bavure_P279 :=[[83.5047578125,129.5107421875,23],[0.330579518507905,-0.31045674667297,-0.610128270725446,0.649674752202896],[0,0,0,0],[8.999999E+09,8.999999E+09,8.999999E+09,8.999999E+09,8.999999E+09,8.999999E+09]];
	LOCAL CONST Robtarget Tr_meulage_bavure_P280 :=[[86.985078125,124.6110859375,23],[0.331182984263124,-0.312332013857537,-0.610884665620476,0.647754945457019],[0,0,0,0],[8.999999E+09,8.999999E+09,8.999999E+09,8.999999E+09,8.999999E+09,8.999999E+09]];
	LOCAL CONST Robtarget Tr_meulage_bavure_P281 :=[[88.3161328125,122.7782578125,23],[0.331854984744675,-0.314258300638438,-0.611577659109389,0.645822542544182],[0,0,0,0],[8.999999E+09,8.999999E+09,8.999999E+09,8.999999E+09,8.999999E+09,8.999999E+09]];
	LOCAL CONST Robtarget Tr_meulage_bavure_P282 :=[[89.13925,121.580046875,23],[0.332513083134098,-0.316135029216154,-0.612229703556002,0.643947577781676],[0,0,0,0],[8.999999E+09,8.999999E+09,8.999999E+09,8.999999E+09,8.999999E+09,8.999999E+09]];
	LOCAL CONST Robtarget Tr_meulage_bavure_P283 :=[[90.125,120.240234375,23],[0.333140158538252,-0.317939195937787,-0.612845869949036,0.642146589294026],[0,0,0,0],[8.999999E+09,8.999999E+09,8.999999E+09,8.999999E+09,8.999999E+09,8.999999E+09]];
	LOCAL CONST Robtarget Tr_meulage_bavure_P284 :=[[93.7008046875,115.11465625,23],[0.333798296947667,-0.319719468012549,-0.613389198623757,0.640399757760975],[0,0,0,0],[8.999999E+09,8.999999E+09,8.999999E+09,8.999999E+09,8.999999E+09,8.999999E+09]];
	LOCAL CONST Robtarget Tr_meulage_bavure_P285 :=[[97.592375,109.600859375,23],[0.334551678788584,-0.321524903335989,-0.613819183420391,0.638688437988075],[0,0,0,0],[8.999999E+09,8.999999E+09,8.999999E+09,8.999999E+09,8.999999E+09,8.999999E+09]];
	LOCAL CONST Robtarget Tr_meulage_bavure_P286 :=[[98.3441171875,108.5922265625,23],[0.335396196079204,-0.323358565530887,-0.614143327652297,0.637005967675006],[0,0,0,0],[8.999999E+09,8.999999E+09,8.999999E+09,8.999999E+09,8.999999E+09,8.999999E+09]];
	LOCAL CONST Robtarget Tr_meulage_bavure_P287 :=[[101.3733828125,104.270046875,23],[0.336224437900344,-0.325118201297148,-0.614417953610987,0.63540684669304],[0,0,0,0],[8.999999E+09,8.999999E+09,8.999999E+09,8.999999E+09,8.999999E+09,8.999999E+09]];
	LOCAL CONST Robtarget Tr_meulage_bavure_P288 :=[[101.6208828125,103.9079609375,23],[0.336825185596452,-0.326602512881066,-0.614756524119373,0.633998429793288],[0,0,0,0],[8.999999E+09,8.999999E+09,8.999999E+09,8.999999E+09,8.999999E+09,8.999999E+09]];
	LOCAL CONST Robtarget Tr_meulage_bavure_P289 :=[[101.8903828125,103.5191328125,23],[0.336991831093118,-0.327613644751758,-0.615273273857498,0.632885932870729],[0,0,0,0],[8.999999E+09,8.999999E+09,8.999999E+09,8.999999E+09,8.999999E+09,8.999999E+09]];
	LOCAL CONST Robtarget Tr_meulage_bavure_P290 :=[[102.08990625,103.272890625,23],[0.33658348293891,-0.328019779593931,-0.616051723846275,0.632135157030436],[0,0,0,0],[8.999999E+09,8.999999E+09,8.999999E+09,8.999999E+09,8.999999E+09,8.999999E+09]];
	LOCAL CONST Robtarget Tr_meulage_bavure_P291 :=[[104.482359375,99.9998203125,23],[0.335585518847736,-0.327816550190742,-0.617111915048461,0.631736933593373],[0,0,0,0],[8.999999E+09,8.999999E+09,8.999999E+09,8.999999E+09,8.999999E+09,8.999999E+09]];
	LOCAL CONST Robtarget Tr_meulage_bavure_P292 :=[[106.0242890625,97.794828125,23],[0.334112456004389,-0.32711698602203,-0.618398069105569,0.631622650262862],[0,0,0,0],[8.999999E+09,8.999999E+09,8.999999E+09,8.999999E+09,8.999999E+09,8.999999E+09]];
	LOCAL CONST Robtarget Tr_meulage_bavure_P293 :=[[108.8211640625,93.874515625,23],[0.332341298396202,-0.326102707101759,-0.619825077332649,0.631682799600248],[0,0,0,0],[8.999999E+09,8.999999E+09,8.999999E+09,8.999999E+09,8.999999E+09,8.999999E+09]];
	LOCAL CONST Robtarget Tr_meulage_bavure_P294 :=[[113.3923359375,87.0133671875,23],[0.330480238690395,-0.32498766811156,-0.621292190578271,0.631792561951313],[0,0,0,0],[8.999999E+09,8.999999E+09,8.999999E+09,8.999999E+09,8.999999E+09,8.999999E+09]];
	LOCAL CONST Robtarget Tr_meulage_bavure_P295 :=[[115.48321875,83.7469140625,23],[0.328724561779311,-0.323966373393537,-0.622700623758784,0.631846408997995],[0,0,0,0],[8.999999E+09,8.999999E+09,8.999999E+09,8.999999E+09,8.999999E+09,8.999999E+09]];
	LOCAL CONST Robtarget Tr_meulage_bavure_P296 :=[[117.0156875,81.979703125,23],[0.327245776290234,-0.323212014404884,-0.623965393535559,0.6317526282609],[0,0,0,0],[8.999999E+09,8.999999E+09,8.999999E+09,8.999999E+09,8.999999E+09,8.999999E+09]];
	LOCAL CONST Robtarget Tr_meulage_bavure_P297 :=[[118.995609375,79.3265078125,23],[0.326156133020319,-0.32284320887683,-0.625034183561592,0.631448104561917],[0,0,0,0],[8.999999E+09,8.999999E+09,8.999999E+09,8.999999E+09,8.999999E+09,8.999999E+09]];
	LOCAL CONST Robtarget Tr_meulage_bavure_P298 :=[[125.1668125,70.38915625,23],[0.325473423868864,-0.32288134313017,-0.625899166281038,0.630923864077306],[0,0,0,0],[8.999999E+09,8.999999E+09,8.999999E+09,8.999999E+09,8.999999E+09,8.999999E+09]];
	LOCAL CONST Robtarget Tr_meulage_bavure_P299 :=[[125.3333125,70.1656796875,23],[0.32513283068146,-0.323261765841991,-0.626590908217328,0.630217666284565],[0,0,0,0],[8.999999E+09,8.999999E+09,8.999999E+09,8.999999E+09,8.999999E+09,8.999999E+09]];
	LOCAL CONST Robtarget Tr_meulage_bavure_P300 :=[[125.586609375,69.796390625,23],[0.325011884371141,-0.323859690665362,-0.627167615551529,0.629398886067544],[0,0,0,0],[8.999999E+09,8.999999E+09,8.999999E+09,8.999999E+09,8.999999E+09,8.999999E+09]];
	LOCAL CONST Robtarget Tr_meulage_bavure_P301 :=[[125.7717890625,69.523921875,23],[0.324966602565154,-0.324532631890869,-0.627702484611466,0.62854185928054],[0,0,0,0],[8.999999E+09,8.999999E+09,8.999999E+09,8.999999E+09,8.999999E+09,8.999999E+09]];
	LOCAL CONST Robtarget Tr_meulage_bavure_P302 :=[[130.5167265625,62.836515625,23],[0.324902229983714,-0.325178316608976,-0.628238615780332,0.627705221422743],[0,0,0,0],[8.999999E+09,8.999999E+09,8.999999E+09,8.999999E+09,8.999999E+09,8.999999E+09]];
	LOCAL CONST Robtarget Tr_meulage_bavure_P303 :=[[133.372921875,58.8506171875,23],[0.324771159020459,-0.325743080537746,-0.628796886120412,0.626920741207021],[0,0,0,0],[8.999999E+09,8.999999E+09,8.999999E+09,8.999999E+09,8.999999E+09,8.999999E+09]];
	LOCAL CONST Robtarget Tr_meulage_bavure_P304 :=[[136.74334375,54.0690625,23],[0.324577902310795,-0.326226856556563,-0.6293724950392,0.626191253436903],[0,0,0,0],[8.999999E+09,8.999999E+09,8.999999E+09,8.999999E+09,8.999999E+09,8.999999E+09]];
	LOCAL CONST Robtarget Tr_meulage_bavure_P305 :=[[140.29046875,49.01486328125,23],[0.324368520398456,-0.326665413860165,-0.629934705928508,0.625505424939582],[0,0,0,0],[8.999999E+09,8.999999E+09,8.999999E+09,8.999999E+09,8.999999E+09,8.999999E+09]];
	LOCAL CONST Robtarget Tr_meulage_bavure_P306 :=[[141.561703125,47.2188125,23],[0.324213443818923,-0.32712303609414,-0.630442337565964,0.624834875073399],[0,0,0,0],[8.999999E+09,8.999999E+09,8.999999E+09,8.999999E+09,8.999999E+09,8.999999E+09]];
	LOCAL CONST Robtarget Tr_meulage_bavure_P307 :=[[141.843078125,46.70169140625,23],[0.324230183755937,-0.327710887107754,-0.630828349799665,0.624128156312205],[0,0,0,0],[8.999999E+09,8.999999E+09,8.999999E+09,8.999999E+09,8.999999E+09,8.999999E+09]];
	LOCAL CONST Robtarget Tr_meulage_bavure_P308 :=[[143.2835625,44.6535625,23],[0.32453058094742,-0.328540027414894,-0.631031374557689,0.623330375274609],[0,0,0,0],[8.999999E+09,8.999999E+09,8.999999E+09,8.999999E+09,8.999999E+09,8.999999E+09]];
	LOCAL CONST Robtarget Tr_meulage_bavure_P309 :=[[147.560296875,38.7595234375,23],[0.325190823182034,-0.329683250752942,-0.631006036631246,0.622407635256903],[0,0,0,0],[8.999999E+09,8.999999E+09,8.999999E+09,8.999999E+09,8.999999E+09,8.999999E+09]];
	LOCAL CONST Robtarget Tr_meulage_bavure_P310 :=[[148.5834375,37.3789375,23],[0.326203147609157,-0.331129528812822,-0.630751390363385,0.62136738343168],[0,0,0,0],[8.999999E+09,8.999999E+09,8.999999E+09,8.999999E+09,8.999999E+09,8.999999E+09]];
	LOCAL CONST Robtarget Tr_meulage_bavure_P311 :=[[149.413578125,36.21926953125,23],[0.327428685443628,-0.332735843125908,-0.630337594579386,0.620283670192778],[0,0,0,0],[8.999999E+09,8.999999E+09,8.999999E+09,8.999999E+09,8.999999E+09,8.999999E+09]];
	LOCAL CONST Robtarget Tr_meulage_bavure_P312 :=[[152.1715625,32.048126953125,23],[0.328610790019844,-0.334244012802049,-0.629903764559596,0.6192876036077],[0,0,0,0],[8.999999E+09,8.999999E+09,8.999999E+09,8.999999E+09,8.999999E+09,8.999999E+09]];
	LOCAL CONST Robtarget Tr_meulage_bavure_P313 :=[[154.777828125,28.24353125,23],[0.329441989073604,-0.335340992641115,-0.629618374802963,0.61854272010927],[0,0,0,0],[8.999999E+09,8.999999E+09,8.999999E+09,8.999999E+09,8.999999E+09,8.999999E+09]];
	LOCAL CONST Robtarget Tr_meulage_bavure_P314 :=[[156.174984375,26.306365234375,23],[0.329660381905224,-0.335759650732623,-0.629627453499624,0.618189905564291],[0,0,0,0],[8.999999E+09,8.999999E+09,8.999999E+09,8.999999E+09,8.999999E+09,8.999999E+09]];
	LOCAL CONST Robtarget Tr_meulage_bavure_P315 :=[[156.5805,25.673919921875,23],[0.32914141568416,-0.335375241142711,-0.63000286838326,0.618292618376413],[0,0,0,0],[8.999999E+09,8.999999E+09,8.999999E+09,8.999999E+09,8.999999E+09,8.999999E+09]];
	LOCAL CONST Robtarget Tr_meulage_bavure_P316 :=[[157.399171875,24.58123828125,23],[0.32794461118741,-0.334256111600229,-0.630716326695853,0.618806996639763],[0,0,0,0],[8.999999E+09,8.999999E+09,8.999999E+09,8.999999E+09,8.999999E+09,8.999999E+09]];
	LOCAL CONST Robtarget Tr_meulage_bavure_P317 :=[[160.299625,20.563384765625,23],[0.326296762371226,-0.332638754405107,-0.631644812775225,0.619602059735138],[0,0,0,0],[8.999999E+09,8.999999E+09,8.999999E+09,8.999999E+09,8.999999E+09,8.999999E+09]];
	LOCAL CONST Robtarget Tr_meulage_bavure_P318 :=[[164.168703125,15.06378125,23],[0.324521644668049,-0.330859014895294,-0.632614545285179,0.62049726147509],[0,0,0,0],[8.999999E+09,8.999999E+09,8.999999E+09,8.999999E+09,8.999999E+09,8.999999E+09]];
	LOCAL CONST Robtarget Tr_meulage_bavure_P319 :=[[165.982546875,12.566345703125,23],[0.322931238704656,-0.329243328587168,-0.633463852284219,0.621319397330193],[0,0,0,0],[8.999999E+09,8.999999E+09,8.999999E+09,8.999999E+09,8.999999E+09,8.999999E+09]];
	LOCAL CONST Robtarget Tr_meulage_bavure_P320 :=[[166.981390625,11.069244140625,23],[0.321754843526292,-0.328036238206497,-0.63408052669165,0.621938849695966],[0,0,0,0],[8.999999E+09,8.999999E+09,8.999999E+09,8.999999E+09,8.999999E+09,8.999999E+09]];
	LOCAL CONST Robtarget Tr_meulage_bavure_P321 :=[[169.84740625,6.9780576171875,23],[0.321108756239763,-0.327363659474308,-0.634411328392047,0.622289697431655],[0,0,0,0],[8.999999E+09,8.999999E+09,8.999999E+09,8.999999E+09,8.999999E+09,8.999999E+09]];
	LOCAL CONST Robtarget Tr_meulage_bavure_P322 :=[[171.244140625,5.03375244140625,23],[0.320983617785543,-0.327220637047497,-0.634466516638367,0.622373208829165],[0,0,0,0],[8.999999E+09,8.999999E+09,8.999999E+09,8.999999E+09,8.999999E+09,8.999999E+09]];
	LOCAL CONST Robtarget Tr_meulage_bavure_P323 :=[[174.20934375,0.91748046875,23],[0.321275790560514,-0.327512776220927,-0.634308893459627,0.622229439587844],[0,0,0,0],[8.999999E+09,8.999999E+09,8.999999E+09,8.999999E+09,8.999999E+09,8.999999E+09]];
	LOCAL CONST Robtarget Tr_meulage_bavure_P324 :=[[178.679203125,-5.309966796875,23],[0.321795219783817,-0.328055258551838,-0.634044082308927,0.621945082422719],[0,0,0,0],[8.999999E+09,8.999999E+09,8.999999E+09,8.999999E+09,8.999999E+09,8.999999E+09]];
	LOCAL CONST Robtarget Tr_meulage_bavure_P325 :=[[179.302984375,-6.1827392578125,23],[0.322293713100575,-0.328596989540904,-0.633803746065991,0.621645873816609],[0,0,0,0],[8.999999E+09,8.999999E+09,8.999999E+09,8.999999E+09,8.999999E+09,8.999999E+09]];
	LOCAL CONST Robtarget Tr_meulage_bavure_P326 :=[[180.069640625,-7.189849609375,23],[0.322513623444945,-0.32888090102587,-0.633728064370305,0.621458812844657],[0,0,0,0],[8.999999E+09,8.999999E+09,8.999999E+09,8.999999E+09,8.999999E+09,8.999999E+09]];
	LOCAL CONST Robtarget Tr_meulage_bavure_P327 :=[[184.452203125,-13.6511533203125,23],[0.322255699008196,-0.328709777529717,-0.633927071945028,0.621480179948087],[0,0,0,0],[8.999999E+09,8.999999E+09,8.999999E+09,8.999999E+09,8.999999E+09,8.999999E+09]];
	LOCAL CONST Robtarget Tr_meulage_bavure_P328 :=[[186.991328125,-17.48260546875,23],[0.321490930401369,-0.328056737001505,-0.634417858995596,0.621720467062998],[0,0,0,0],[8.999999E+09,8.999999E+09,8.999999E+09,8.999999E+09,8.999999E+09,8.999999E+09]];
	LOCAL CONST Robtarget Tr_meulage_bavure_P329 :=[[189.965328125,-21.880919921875,23],[0.320404434570719,-0.32710913012892,-0.635100804744304,0.622083260590459],[0,0,0,0],[8.999999E+09,8.999999E+09,8.999999E+09,8.999999E+09,8.999999E+09,8.999999E+09]];
	LOCAL CONST Robtarget Tr_meulage_bavure_P330 :=[[192.81275,-26.05471875,23],[0.319380760795688,-0.326261566219921,-0.635774710380086,0.622366321134434],[0,0,0,0],[8.999999E+09,8.999999E+09,8.999999E+09,8.999999E+09,8.999999E+09,8.999999E+09]];
	LOCAL CONST Robtarget Tr_meulage_bavure_P331 :=[[193.543578125,-27.085998046875,23],[0.318962776284457,-0.326070969474194,-0.636157419832983,0.622289488423605],[0,0,0,0],[8.999999E+09,8.999999E+09,8.999999E+09,8.999999E+09,8.999999E+09,8.999999E+09]];
	LOCAL CONST Robtarget Tr_meulage_bavure_P332 :=[[194.673765625,-28.60726953125,23],[0.319723569944138,-0.327121975547774,-0.635946056349961,0.621563082356754],[0,0,0,0],[8.999999E+09,8.999999E+09,8.999999E+09,8.999999E+09,8.999999E+09,8.999999E+09]];
	LOCAL CONST Robtarget Tr_meulage_bavure_P333 :=[[195.8959375,-30.206755859375,23],[0.32222638932699,-0.329992971344416,-0.634831379065299,0.619890242735458],[0,0,0,0],[8.999999E+09,8.999999E+09,8.999999E+09,8.999999E+09,8.999999E+09,8.999999E+09]];
	LOCAL CONST Robtarget Tr_meulage_bavure_P334 :=[[198.542046875,-33.70907421875,23],[0.327017954315916,-0.335250813697078,-0.632484203407469,0.616952090449899],[0,0,0,0],[8.999999E+09,8.999999E+09,8.999999E+09,8.999999E+09,8.999999E+09,8.999999E+09]];
	LOCAL CONST Robtarget Tr_meulage_bavure_P335 :=[[199.99846875,-35.74435546875,23],[0.334550802915428,-0.343364906666801,-0.628569894902319,0.612434640072579],[0,0,0,0],[8.999999E+09,8.999999E+09,8.999999E+09,8.999999E+09,8.999999E+09,8.999999E+09]];
	LOCAL CONST Robtarget Tr_meulage_bavure_P336 :=[[200.7315,-36.8044453125,23],[0.345073548506536,-0.354600900854032,-0.622794117617852,0.60606099882373],[0,0,0,0],[8.999999E+09,8.999999E+09,8.999999E+09,8.999999E+09,8.999999E+09,8.999999E+09]];
	LOCAL CONST Robtarget Tr_meulage_bavure_P337 :=[[202.227421875,-38.6184375,23],[0.35855807500875,-0.368937633166126,-0.614938726348127,0.59763826225999],[0,0,0,0],[8.999999E+09,8.999999E+09,8.999999E+09,8.999999E+09,8.999999E+09,8.999999E+09]];
	LOCAL CONST Robtarget Tr_meulage_bavure_P338 :=[[203.950921875,-40.7932109375,23],[0.374653499026549,-0.386027042443334,-0.604922789128762,0.587099904072805],[0,0,0,0],[8.999999E+09,8.999999E+09,8.999999E+09,8.999999E+09,8.999999E+09,8.999999E+09]];
	LOCAL CONST Robtarget Tr_meulage_bavure_P339 :=[[205.759640625,-43.88290234375,23],[0.392981486742592,-0.405487646346992,-0.592653860684545,0.574375070100769],[0,0,0,0],[8.999999E+09,8.999999E+09,8.999999E+09,8.999999E+09,8.999999E+09,8.999999E+09]];
	LOCAL CONST Robtarget Tr_meulage_bavure_P340 :=[[205.90075,-44.10342578125,23],[0.413562869746439,-0.427346019600313,-0.577721173176452,0.559087988032726],[0,0,0,0],[8.999999E+09,8.999999E+09,8.999999E+09,8.999999E+09,8.999999E+09,8.999999E+09]];
	LOCAL CONST Robtarget Tr_meulage_bavure_P341 :=[[206.1639375,-45.01780859375,23],[0.437013639367846,-0.452246196758434,-0.559104490718601,0.540272732036603],[0,0,0,0],[8.999999E+09,8.999999E+09,8.999999E+09,8.999999E+09,8.999999E+09,8.999999E+09]];
	LOCAL CONST Robtarget Tr_meulage_bavure_P342 :=[[206.448125,-46.1610859375,23],[0.46422078063692,-0.481115334013954,-0.535157740318525,0.516365466679037],[0,0,0,0],[8.999999E+09,8.999999E+09,8.999999E+09,8.999999E+09,8.999999E+09,8.999999E+09]];
	LOCAL CONST Robtarget Tr_meulage_bavure_P343 :=[[206.25659375,-46.800046875,23],[0.495364466641452,-0.514151437141929,-0.504233812299886,0.485809229438308],[0,0,0,0],[8.999999E+09,8.999999E+09,8.999999E+09,8.999999E+09,8.999999E+09,8.999999E+09]];
	LOCAL CONST Robtarget Tr_meulage_bavure_P344 :=[[205.84784375,-47.54510546875,23],[0.528898856976665,-0.549760030484462,-0.465936256340578,0.448255856624125],[0,0,0,0],[8.999999E+09,8.999999E+09,8.999999E+09,8.999999E+09,8.999999E+09,8.999999E+09]];
	LOCAL CONST Robtarget Tr_meulage_bavure_P345 :=[[205.15984375,-49.511,23],[0.56152742688184,-0.584502450205446,-0.422369888290514,0.405767805559718],[0,0,0,0],[8.999999E+09,8.999999E+09,8.999999E+09,8.999999E+09,8.999999E+09,8.999999E+09]];
	LOCAL CONST Robtarget Tr_meulage_bavure_P346 :=[[203.30071875,-51.18824609375,23],[0.589938581284223,-0.614913102055539,-0.377625832390185,0.362288666596697],[0,0,0,0],[8.999999E+09,8.999999E+09,8.999999E+09,8.999999E+09,8.999999E+09,8.999999E+09]];
	LOCAL CONST Robtarget Tr_meulage_bavure_P347 :=[[203.253109375,-51.2399296875,23],[0.612691686728111,-0.639456826456782,-0.335351422511645,0.321314935120514],[0,0,0,0],[8.999999E+09,8.999999E+09,8.999999E+09,8.999999E+09,8.999999E+09,8.999999E+09]];
	LOCAL CONST Robtarget Tr_meulage_bavure_P348 :=[[203.158265625,-51.3037109375,23],[0.630311515766614,-0.658643238909082,-0.296915569645253,0.284143663370453],[0,0,0,0],[8.999999E+09,8.999999E+09,8.999999E+09,8.999999E+09,8.999999E+09,8.999999E+09]];
	LOCAL CONST Robtarget Tr_meulage_bavure_P349 :=[[202.124265625,-51.73040625,23],[0.644063698326776,-0.673763535449376,-0.261855361783178,0.25031264510966],[0,0,0,0],[8.999999E+09,8.999999E+09,8.999999E+09,8.999999E+09,8.999999E+09,8.999999E+09]];
	LOCAL CONST Robtarget Tr_meulage_bavure_P350 :=[[200.7029375,-52.2183984375,23],[0.65499003279361,-0.685881364441163,-0.22933116550951,0.219002345602518],[0,0,0,0],[8.999999E+09,8.999999E+09,8.999999E+09,8.999999E+09,8.999999E+09,8.999999E+09]];
	LOCAL CONST Robtarget Tr_meulage_bavure_P351 :=[[198.012640625,-53.244765625,23],[0.663599877227408,-0.695504406176502,-0.199337315602008,0.190193213710229],[0,0,0,0],[8.999999E+09,8.999999E+09,8.999999E+09,8.999999E+09,8.999999E+09,8.999999E+09]];
	LOCAL CONST Robtarget Tr_meulage_bavure_P352 :=[[193.5468125,-54.7698359375,23],[0.670094006631479,-0.702820968267198,-0.172819913618464,0.164772528952603],[0,0,0,0],[8.999999E+09,8.999999E+09,8.999999E+09,8.999999E+09,8.999999E+09,8.999999E+09]];
	LOCAL CONST Robtarget Tr_meulage_bavure_P353 :=[[192.344671875,-55.2086796875,23],[0.674675781600523,-0.708025926234832,-0.151012633645986,0.143899485684747],[0,0,0,0],[8.999999E+09,8.999999E+09,8.999999E+09,8.999999E+09,8.999999E+09,8.999999E+09]];
	LOCAL CONST Robtarget Tr_meulage_bavure_P354 :=[[191.9919375,-55.328796875,23],[0.677680487668268,-0.711459043687216,-0.134639638486402,0.128247235984336],[0,0,0,0],[8.999999E+09,8.999999E+09,8.999999E+09,8.999999E+09,8.999999E+09,8.999999E+09]];
	LOCAL CONST Robtarget Tr_meulage_bavure_P355 :=[[186.362796875,-57.39591796875,23],[0.6795223939019,-0.713527585114849,-0.123589854291533,0.117699827451873],[0,0,0,0],[8.999999E+09,8.999999E+09,8.999999E+09,8.999999E+09,8.999999E+09,8.999999E+09]];
	LOCAL CONST Robtarget Tr_meulage_bavure_P356 :=[[182.713015625,-58.45585546875,23],[0.680572857165536,-0.714606948778984,-0.117117271509603,0.111539408105272],[0,0,0,0],[8.999999E+09,8.999999E+09,8.999999E+09,8.999999E+09,8.999999E+09,8.999999E+09]];
	LOCAL CONST Robtarget Tr_meulage_bavure_P357 :=[[181.017390625,-58.9974375,23],[0.681124607458308,-0.714991544447041,-0.114152487330202,0.108745437239129],[0,0,0,0],[8.999999E+09,8.999999E+09,8.999999E+09,8.999999E+09,8.999999E+09,8.999999E+09]];
	LOCAL CONST Robtarget Tr_meulage_bavure_P358 :=[[179.954953125,-59.32169921875,23],[0.681398867650114,-0.714899420954388,-0.113566806144333,0.108245007397098],[0,0,0,0],[8.999999E+09,8.999999E+09,8.999999E+09,8.999999E+09,8.999999E+09,8.999999E+09]];
	LOCAL CONST Robtarget Tr_meulage_bavure_P359 :=[[178.469421875,-59.82896484375,23],[0.681561026561449,-0.714489753578789,-0.114360535303839,0.109089995271999],[0,0,0,0],[8.999999E+09,8.999999E+09,8.999999E+09,8.999999E+09,8.999999E+09,8.999999E+09]];
	LOCAL CONST Robtarget Tr_meulage_bavure_P360 :=[[176.7160625,-60.41717578125,23],[0.68174214070192,-0.713888358624534,-0.115692139135705,0.110482550449099],[0,0,0,0],[8.999999E+09,8.999999E+09,8.999999E+09,8.999999E+09,8.999999E+09,8.999999E+09]];
	LOCAL CONST Robtarget Tr_meulage_bavure_P361 :=[[175.736203125,-60.8102109375,23],[0.682049871229227,-0.713197487106037,-0.116885867379151,0.11178108761706],[0,0,0,0],[8.999999E+09,8.999999E+09,8.999999E+09,8.999999E+09,8.999999E+09,8.999999E+09]];
	LOCAL CONST Robtarget Tr_meulage_bavure_P362 :=[[170.52625,-62.6911171875,23],[0.68254637612051,-0.712481785933725,-0.117551988752475,0.112612961499937],[0,0,0,0],[8.999999E+09,8.999999E+09,8.999999E+09,8.999999E+09,8.999999E+09,8.999999E+09]];
	LOCAL CONST Robtarget Tr_meulage_bavure_P363 :=[[169.945796875,-62.88107421875,23],[0.683255756403071,-0.711762626553105,-0.117559333727616,0.112850954084634],[0,0,0,0],[8.999999E+09,8.999999E+09,8.999999E+09,8.999999E+09,8.999999E+09,8.999999E+09]];
	LOCAL CONST Robtarget Tr_meulage_bavure_P364 :=[[167.422,-63.584625,23],[0.684160028775934,-0.711027975559473,-0.117002822267397,0.112581581879871],[0,0,0,0],[8.999999E+09,8.999999E+09,8.999999E+09,8.999999E+09,8.999999E+09,8.999999E+09]];
	LOCAL CONST Robtarget Tr_meulage_bavure_P365 :=[[166.197140625,-63.8701640625,23],[0.685214434233059,-0.710246143216314,-0.116114602701912,0.112022293336629],[0,0,0,0],[8.999999E+09,8.999999E+09,8.999999E+09,8.999999E+09,8.999999E+09,8.999999E+09]];
	LOCAL CONST Robtarget Tr_meulage_bavure_P366 :=[[165.289984375,-64.1312265625,23],[0.686371144043042,-0.709387446598694,-0.115130978042672,0.111395516643033],[0,0,0,0],[8.999999E+09,8.999999E+09,8.999999E+09,8.999999E+09,8.999999E+09,8.999999E+09]];
	LOCAL CONST Robtarget Tr_meulage_bavure_P367 :=[[163.7109375,-64.62452734375,23],[0.687597806035143,-0.708440292855968,-0.11418741218223,0.110827990566165],[0,0,0,0],[8.999999E+09,8.999999E+09,8.999999E+09,8.999999E+09,8.999999E+09,8.999999E+09]];
	LOCAL CONST Robtarget Tr_meulage_bavure_P368 :=[[156.487359375,-67.03453125,23],[0.68887313660506,-0.707421478065288,-0.113298202616933,0.110327563734557],[0,0,0,0],[8.999999E+09,8.999999E+09,8.999999E+09,8.999999E+09,8.999999E+09,8.999999E+09]];
	LOCAL CONST Robtarget Tr_meulage_bavure_P369 :=[[155.624515625,-67.3116328125,23],[0.690185156029896,-0.706357653652406,-0.11241749510073,0.109843626660509],[0,0,0,0],[8.999999E+09,8.999999E+09,8.999999E+09,8.999999E+09,8.999999E+09,8.999999E+09]];
	LOCAL CONST Robtarget Tr_meulage_bavure_P370 :=[[155.4138125,-67.382296875,23],[0.691512238195941,-0.70527455692011,-0.111533332811704,0.10935693603195],[0,0,0,0],[8.999999E+09,8.999999E+09,8.999999E+09,8.999999E+09,8.999999E+09,8.999999E+09]];
	LOCAL CONST Robtarget Tr_meulage_bavure_P371 :=[[155.090390625,-67.485109375,23],[0.692822876064291,-0.704180681409283,-0.110721044532689,0.108935212991727],[0,0,0,0],[8.999999E+09,8.999999E+09,8.999999E+09,8.999999E+09,8.999999E+09,8.999999E+09]];
	LOCAL CONST Robtarget Tr_meulage_bavure_P372 :=[[150.60053125,-68.875796875,23],[0.694067781530484,-0.703071446771659,-0.110157301282039,0.108746606154013],[0,0,0,0],[8.999999E+09,8.999999E+09,8.999999E+09,8.999999E+09,8.999999E+09,8.999999E+09]];
	LOCAL CONST Robtarget Tr_meulage_bavure_P373 :=[[148.522828125,-69.4526640625,23],[0.695189786923288,-0.701946305314957,-0.110032943405823,0.108973831618808],[0,0,0,0],[8.999999E+09,8.999999E+09,8.999999E+09,8.999999E+09,8.999999E+09,8.999999E+09]];
	LOCAL CONST Robtarget Tr_meulage_bavure_P374 :=[[140.532890625,-71.55284375,23],[0.69615251664004,-0.700810169727667,-0.110449977048212,0.109715915673465],[0,0,0,0],[8.999999E+09,8.999999E+09,8.999999E+09,8.999999E+09,8.999999E+09,8.999999E+09]];
	LOCAL CONST Robtarget Tr_meulage_bavure_P375 :=[[138.825140625,-72.09296875,23],[0.696940183241611,-0.699689612269367,-0.111369007177619,0.110931382871416],[0,0,0,0],[8.999999E+09,8.999999E+09,8.999999E+09,8.999999E+09,8.999999E+09,8.999999E+09]];
	LOCAL CONST Robtarget Tr_meulage_bavure_P376 :=[[135.917484375,-73.0869765625,23],[0.697558866317387,-0.698630401403867,-0.112618972675114,0.112446241599595],[0,0,0,0],[8.999999E+09,8.999999E+09,8.999999E+09,8.999999E+09,8.999999E+09,8.999999E+09]];
	LOCAL CONST Robtarget Tr_meulage_bavure_P377 :=[[134.714359375,-73.4005546875,23],[0.698031853547371,-0.697688406970285,-0.113950934974107,0.114007028866712],[0,0,0,0],[8.999999E+09,8.999999E+09,8.999999E+09,8.999999E+09,8.999999E+09,8.999999E+09]];
	LOCAL CONST Robtarget Tr_meulage_bavure_P378 :=[[132.3591875,-73.9639140625,23],[0.698400543205327,-0.696919141690587,-0.115073966973447,0.115318573182093],[0,0,0,0],[8.999999E+09,8.999999E+09,8.999999E+09,8.999999E+09,8.999999E+09,8.999999E+09]];
	LOCAL CONST Robtarget Tr_meulage_bavure_P379 :=[[129.667171875,-74.7458515625,23],[0.698702302116262,-0.696384806266303,-0.115702301479444,0.116087346645703],[0,0,0,0],[8.999999E+09,8.999999E+09,8.999999E+09,8.999999E+09,8.999999E+09,8.999999E+09]];
	LOCAL CONST Robtarget Tr_meulage_bavure_P380 :=[[126.146421875,-75.689546875,23],[0.698977524154344,-0.696134938723649,-0.115579514450663,0.116051469851245],[0,0,0,0],[8.999999E+09,8.999999E+09,8.999999E+09,8.999999E+09,8.999999E+09,8.999999E+09]];
	LOCAL CONST Robtarget Tr_meulage_bavure_P381 :=[[125.0880703125,-75.991609375,23],[0.699248709425611,-0.696190677122777,-0.114573574639518,0.115076841494149],[0,0,0,0],[8.999999E+09,8.999999E+09,8.999999E+09,8.999999E+09,8.999999E+09,8.999999E+09]];
	LOCAL CONST Robtarget Tr_meulage_bavure_P382 :=[[119.507015625,-78.2035078125,23],[0.699504392310141,-0.696532020106434,-0.112756390968691,0.113237566209212],[0,0,0,0],[8.999999E+09,8.999999E+09,8.999999E+09,8.999999E+09,8.999999E+09,8.999999E+09]];
	LOCAL CONST Robtarget Tr_meulage_bavure_P383 :=[[118.90509375,-78.42375,23],[0.699686372188468,-0.697092041419977,-0.110477711510577,0.110888870595997],[0,0,0,0],[8.999999E+09,8.999999E+09,8.999999E+09,8.999999E+09,8.999999E+09,8.999999E+09]];
	LOCAL CONST Robtarget Tr_meulage_bavure_P384 :=[[117.274171875,-78.9854453125,23],[0.699708911454338,-0.697769192028768,-0.108305785387607,0.108606863219959],[0,0,0,0],[8.999999E+09,8.999999E+09,8.999999E+09,8.999999E+09,8.999999E+09,8.999999E+09]];
	LOCAL CONST Robtarget Tr_meulage_bavure_P385 :=[[116.2760625,-79.329484375,23],[0.699489233647061,-0.698462170199821,-0.106845240353897,0.107002352428911],[0,0,0,0],[8.999999E+09,8.999999E+09,8.999999E+09,8.999999E+09,8.999999E+09,8.999999E+09]];
	LOCAL CONST Robtarget Tr_meulage_bavure_P386 :=[[116.14196875,-79.363828125,23],[0.698977380563461,-0.699092530613392,-0.106545751792273,0.106528202257553],[0,0,0,0],[8.999999E+09,8.999999E+09,8.999999E+09,8.999999E+09,8.999999E+09,8.999999E+09]];
	LOCAL CONST Robtarget Tr_meulage_bavure_P387 :=[[115.961,-79.415484375,23],[0.698168751943993,-0.699624329272431,-0.107550622451757,0.107326862011832],[0,0,0,0],[8.999999E+09,8.999999E+09,8.999999E+09,8.999999E+09,8.999999E+09,8.999999E+09]];
	LOCAL CONST Robtarget Tr_meulage_bavure_P388 :=[[113.60796875,-79.9984609375,23],[0.69710067095522,-0.70006758990346,-0.109676264521005,0.109211451419995],[0,0,0,0],[8.999999E+09,8.999999E+09,8.999999E+09,8.999999E+09,8.999999E+09,8.999999E+09]];
	LOCAL CONST Robtarget Tr_meulage_bavure_P389 :=[[110.2039765625,-80.848828125,23],[0.695842696571006,-0.700458126510866,-0.11253375716317,0.111792254348943],[0,0,0,0],[8.999999E+09,8.999999E+09,8.999999E+09,8.999999E+09,8.999999E+09,8.999999E+09]];
	LOCAL CONST Robtarget Tr_meulage_bavure_P390 :=[[106.754390625,-82.0574609375,23],[0.69446875956046,-0.700843621120534,-0.115701743822138,0.114649322744315],[0,0,0,0],[8.999999E+09,8.999999E+09,8.999999E+09,8.999999E+09,8.999999E+09,8.999999E+09]];
	LOCAL CONST Robtarget Tr_meulage_bavure_P391 :=[[105.112546875,-82.6219140625,23],[0.693052656743597,-0.701263749180236,-0.118818868090931,0.11742761877817],[0,0,0,0],[8.999999E+09,8.999999E+09,8.999999E+09,8.999999E+09,8.999999E+09,8.999999E+09]];
	LOCAL CONST Robtarget Tr_meulage_bavure_P392 :=[[103.1006171875,-83.3198515625,23],[0.691651511643508,-0.701753255801914,-0.121621013393246,0.119870277858459],[0,0,0,0],[8.999999E+09,8.999999E+09,8.999999E+09,8.999999E+09,8.999999E+09,8.999999E+09]];
	LOCAL CONST Robtarget Tr_meulage_bavure_P393 :=[[99.558109375,-84.4078671875,23],[0.690324376509229,-0.702348052750034,-0.123855146031428,0.121734838057613],[0,0,0,0],[8.999999E+09,8.999999E+09,8.999999E+09,8.999999E+09,8.999999E+09,8.999999E+09]];
	LOCAL CONST Robtarget Tr_meulage_bavure_P394 :=[[94.443515625,-86.0073125,23],[0.689142649420193,-0.703097075207965,-0.125205834790565,0.122720864234737],[0,0,0,0],[8.999999E+09,8.999999E+09,8.999999E+09,8.999999E+09,8.999999E+09,8.999999E+09]];
	LOCAL CONST Robtarget Tr_meulage_bavure_P395 :=[[93.7944375,-86.2887578125,23],[0.688187435734997,-0.704060181278451,-0.125293997753493,0.1224692964036],[0,0,0,0],[8.999999E+09,8.999999E+09,8.999999E+09,8.999999E+09,8.999999E+09,8.999999E+09]];
	LOCAL CONST Robtarget Tr_meulage_bavure_P396 :=[[93.4739375,-86.409453125,23],[0.687519155202576,-0.705283197304922,-0.123805129896498,0.12068683706268],[0,0,0,0],[8.999999E+09,8.999999E+09,8.999999E+09,8.999999E+09,8.999999E+09,8.999999E+09]];
	LOCAL CONST Robtarget Tr_meulage_bavure_P397 :=[[91.8763125,-87.058109375,23],[0.687144178124598,-0.706750426792802,-0.120693231628797,0.11734503200673],[0,0,0,0],[8.999999E+09,8.999999E+09,8.999999E+09,8.999999E+09,8.999999E+09,8.999999E+09]];
	LOCAL CONST Robtarget Tr_meulage_bavure_P398 :=[[89.365203125,-88.0823359375,23],[0.68699199696787,-0.708377325349918,-0.116292273892511,0.11278150586467],[0,0,0,0],[8.999999E+09,8.999999E+09,8.999999E+09,8.999999E+09,8.999999E+09,8.999999E+09]];
	LOCAL CONST Robtarget Tr_meulage_bavure_P399 :=[[88.6456875,-88.3218359375,23],[0.6869412985619,-0.710014501184016,-0.111317909887344,0.107700433503386],[0,0,0,0],[8.999999E+09,8.999999E+09,8.999999E+09,8.999999E+09,8.999999E+09,8.999999E+09]];
	LOCAL CONST Robtarget Tr_meulage_bavure_P400 :=[[86.30990625,-89.028125,23],[0.686856807339738,-0.711505863576537,-0.106681839108511,0.102986006387734],[0,0,0,0],[8.999999E+09,8.999999E+09,8.999999E+09,8.999999E+09,8.999999E+09,8.999999E+09]];
	LOCAL CONST Robtarget Tr_meulage_bavure_P401 :=[[83.1664140625,-89.841671875,23],[0.686640174396385,-0.712726589232768,-0.103227507959464,0.099449291128722],[0,0,0,0],[8.999999E+09,8.999999E+09,8.999999E+09,8.999999E+09,8.999999E+09,8.999999E+09]];
	LOCAL CONST Robtarget Tr_meulage_bavure_P402 :=[[81.96740625,-90.194703125,23],[0.686240065075905,-0.713609211368014,-0.10151806563197,0.0976245301432014],[0,0,0,0],[8.999999E+09,8.999999E+09,8.999999E+09,8.999999E+09,8.999999E+09,8.999999E+09]];
	LOCAL CONST Robtarget Tr_meulage_bavure_P403 :=[[77.14053125,-91.469296875,23],[0.685649545564598,-0.714132795051763,-0.101755938242752,0.0976973936753389],[0,0,0,0],[8.999999E+09,8.999999E+09,8.999999E+09,8.999999E+09,8.999999E+09,8.999999E+09]];
	LOCAL CONST Robtarget Tr_meulage_bavure_P404 :=[[75.410921875,-91.9763984375,23],[0.684899496305386,-0.714301160304121,-0.103816011660776,0.0995427951770744],[0,0,0,0],[8.999999E+09,8.999999E+09,8.999999E+09,8.999999E+09,8.999999E+09,8.999999E+09]];
	LOCAL CONST Robtarget Tr_meulage_bavure_P405 :=[[71.5380546875,-92.8167890625,23],[0.684035504611063,-0.714153876015712,-0.107309049323404,0.102783450693829],[0,0,0,0],[8.999999E+09,8.999999E+09,8.999999E+09,8.999999E+09,8.999999E+09,8.999999E+09]];
	LOCAL CONST Robtarget Tr_meulage_bavure_P406 :=[[70.041171875,-93.2783984375,23],[0.68312651220422,-0.713755334852988,-0.111666251657733,0.106874405417337],[0,0,0,0],[8.999999E+09,8.999999E+09,8.999999E+09,8.999999E+09,8.999999E+09,8.999999E+09]];
	LOCAL CONST Robtarget Tr_meulage_bavure_P407 :=[[69.3017265625,-93.53903125,23],[0.682265972271942,-0.713197338368813,-0.116208141356907,0.111168194668423],[0,0,0,0],[8.999999E+09,8.999999E+09,8.999999E+09,8.999999E+09,8.999999E+09,8.999999E+09]];
	LOCAL CONST Robtarget Tr_meulage_bavure_P408 :=[[68.0478203125,-93.966078125,23],[0.681566158190504,-0.712599685386795,-0.120209113276326,0.114974038292988],[0,0,0,0],[8.999999E+09,8.999999E+09,8.999999E+09,8.999999E+09,8.999999E+09,8.999999E+09]];
	LOCAL CONST Robtarget Tr_meulage_bavure_P409 :=[[65.762421875,-94.8878046875,23],[0.681143257227355,-0.712082683391888,-0.123021735335064,0.117676538792857],[0,0,0,0],[8.999999E+09,8.999999E+09,8.999999E+09,8.999999E+09,8.999999E+09,8.999999E+09]];
	LOCAL CONST Robtarget Tr_meulage_bavure_P410 :=[[64.7054140625,-95.309109375,23],[0.681072461133073,-0.711735749908829,-0.124245721503455,0.118892916845124],[0,0,0,0],[8.999999E+09,8.999999E+09,8.999999E+09,8.999999E+09,8.999999E+09,8.999999E+09]];
	LOCAL CONST Robtarget Tr_meulage_bavure_P411 :=[[63.70816015625,-95.8070703125,23],[0.681361775890491,-0.71158336294309,-0.123834924232573,0.118575543339563],[0,0,0,0],[8.999999E+09,8.999999E+09,8.999999E+09,8.999999E+09,8.999999E+09,8.999999E+09]];
	LOCAL CONST Robtarget Tr_meulage_bavure_P412 :=[[61.37555078125,-96.6091484375,23],[0.681944162651622,-0.711577960518078,-0.122117109786415,0.117031519804382],[0,0,0,0],[8.999999E+09,8.999999E+09,8.999999E+09,8.999999E+09,8.999999E+09,8.999999E+09]];
	LOCAL CONST Robtarget Tr_meulage_bavure_P413 :=[[60.29055859375,-97.0237421875,23],[0.682700888809609,-0.71162452198041,-0.119688912636471,0.114824214896608],[0,0,0,0],[8.999999E+09,8.999999E+09,8.999999E+09,8.999999E+09,8.999999E+09,8.999999E+09]];
	LOCAL CONST Robtarget Tr_meulage_bavure_P414 :=[[53.4247734375,-99.0342421875,23],[0.683508173709794,-0.711622642163973,-0.117204462220438,0.112574000848712],[0,0,0,0],[8.999999E+09,8.999999E+09,8.999999E+09,8.999999E+09,8.999999E+09,8.999999E+09]];
	LOCAL CONST Robtarget Tr_meulage_bavure_P415 :=[[52.94098046875,-99.1720859375,23],[0.684274916412267,-0.711504243702899,-0.11516346869565,0.110756153055874],[0,0,0,0],[8.999999E+09,8.999999E+09,8.999999E+09,8.999999E+09,8.999999E+09,8.999999E+09]];
	LOCAL CONST Robtarget Tr_meulage_bavure_P416 :=[[52.7060234375,-99.2255078125,23],[0.684950784968821,-0.711257313677978,-0.113788211439313,0.10957964613752],[0,0,0,0],[8.999999E+09,8.999999E+09,8.999999E+09,8.999999E+09,8.999999E+09,8.999999E+09]];
	LOCAL CONST Robtarget Tr_meulage_bavure_P417 :=[[51.5375078125,-99.6216875,23],[0.685522121455412,-0.710909015666178,-0.113058412173146,0.109021043274698],[0,0,0,0],[8.999999E+09,8.999999E+09,8.999999E+09,8.999999E+09,8.999999E+09,8.999999E+09]];
	LOCAL CONST Robtarget Tr_meulage_bavure_P418 :=[[45.384734375,-101.7522578125,23],[0.685993096902808,-0.710504386532477,-0.112827685540436,0.108935306927513],[0,0,0,0],[8.999999E+09,8.999999E+09,8.999999E+09,8.999999E+09,8.999999E+09,8.999999E+09]];
	LOCAL CONST Robtarget Tr_meulage_bavure_P419 :=[[40.6701953125,-103.2375625,23],[0.686372162308814,-0.710079228504604,-0.112956839776419,0.109185605285465],[0,0,0,0],[8.999999E+09,8.999999E+09,8.999999E+09,8.999999E+09,8.999999E+09,8.999999E+09]];
	LOCAL CONST Robtarget Tr_meulage_bavure_P420 :=[[37.8361796875,-104.09959375,23],[0.686653473405722,-0.709656548833963,-0.113390043611717,0.109714575907942],[0,0,0,0],[8.999999E+09,8.999999E+09,8.999999E+09,8.999999E+09,8.999999E+09,8.999999E+09]];
	LOCAL CONST Robtarget Tr_meulage_bavure_P421 :=[[37.293578125,-104.325484375,23],[0.686818562782276,-0.709250215063796,-0.114139005043964,0.110529099232832],[0,0,0,0],[8.999999E+09,8.999999E+09,8.999999E+09,8.999999E+09,8.999999E+09,8.999999E+09]];
	LOCAL CONST Robtarget Tr_meulage_bavure_P422 :=[[36.0713515625,-104.6773515625,23],[0.686855917644789,-0.708871481434856,-0.115199134402601,0.11162137177789],[0,0,0,0],[8.999999E+09,8.999999E+09,8.999999E+09,8.999999E+09,8.999999E+09,8.999999E+09]];
	LOCAL CONST Robtarget Tr_meulage_bavure_P423 :=[[31.106201171875,-106.3317578125,23],[0.686771666156025,-0.70854131478169,-0.116479142971124,0.11290036787107],[0,0,0,0],[8.999999E+09,8.999999E+09,8.999999E+09,8.999999E+09,8.999999E+09,8.999999E+09]];
	LOCAL CONST Robtarget Tr_meulage_bavure_P424 :=[[30.47784375,-106.539171875,23],[0.686587051485315,-0.70829091009015,-0.1178130015002,0.114202907554414],[0,0,0,0],[8.999999E+09,8.999999E+09,8.999999E+09,8.999999E+09,8.999999E+09,8.999999E+09]];
	LOCAL CONST Robtarget Tr_meulage_bavure_P425 :=[[28.3955078125,-107.2458359375,23],[0.686330385721612,-0.708158454716291,-0.118999435190285,0.115331431420279],[0,0,0,0],[8.999999E+09,8.999999E+09,8.999999E+09,8.999999E+09,8.999999E+09,8.999999E+09]];
	LOCAL CONST Robtarget Tr_meulage_bavure_P426 :=[[24.538177734375,-108.52359375,23],[0.686027198254287,-0.708164561698731,-0.11990508199107,0.116156825551203],[0,0,0,0],[8.999999E+09,8.999999E+09,8.999999E+09,8.999999E+09,8.999999E+09,8.999999E+09]];
	LOCAL CONST Robtarget Tr_meulage_bavure_P427 :=[[23.168517578125,-108.9599140625,23],[0.68567744599676,-0.708302638544607,-0.120555963189661,0.11670506424968],[0,0,0,0],[8.999999E+09,8.999999E+09,8.999999E+09,8.999999E+09,8.999999E+09,8.999999E+09]];
	LOCAL CONST Robtarget Tr_meulage_bavure_P428 :=[[20.88366796875,-109.7016484375,23],[0.68525172327249,-0.708538353504439,-0.121145181329068,0.11716365650682],[0,0,0,0],[8.999999E+09,8.999999E+09,8.999999E+09,8.999999E+09,8.999999E+09,8.999999E+09]];
	LOCAL CONST Robtarget Tr_meulage_bavure_P429 :=[[17.02209375,-111.034515625,23],[0.68470778587979,-0.70881463357319,-0.121966624365598,0.117818528801547],[0,0,0,0],[8.999999E+09,8.999999E+09,8.999999E+09,8.999999E+09,8.999999E+09,8.999999E+09]];
	LOCAL CONST Robtarget Tr_meulage_bavure_P430 :=[[14.5592041015625,-111.8954140625,23],[0.684011088606804,-0.70907178751878,-0.123291368517773,0.118933886074872],[0,0,0,0],[8.999999E+09,8.999999E+09,8.999999E+09,8.999999E+09,8.999999E+09,8.999999E+09]];
	LOCAL CONST Robtarget Tr_meulage_bavure_P431 :=[[11.2615048828125,-112.957125,23],[0.68314606435333,-0.709274274045075,-0.125251740849425,0.120637723580047],[0,0,0,0],[8.999999E+09,8.999999E+09,8.999999E+09,8.999999E+09,8.999999E+09,8.999999E+09]];
	LOCAL CONST Robtarget Tr_meulage_bavure_P432 :=[[8.704833984375,-113.731078125,23],[0.682124670021308,-0.709417614882541,-0.127798886648686,0.122882166379192],[0,0,0,0],[8.999999E+09,8.999999E+09,8.999999E+09,8.999999E+09,8.999999E+09,8.999999E+09]];
	LOCAL CONST Robtarget Tr_meulage_bavure_P433 :=[[7.0339052734375,-114.249265625,23],[0.680986264774851,-0.709520570010243,-0.130739120637825,0.125481274520083],[0,0,0,0],[8.999999E+09,8.999999E+09,8.999999E+09,8.999999E+09,8.999999E+09,8.999999E+09]];
	LOCAL CONST Robtarget Tr_meulage_bavure_P434 :=[[3.26043701171875,-115.742890625,23],[0.679775108541029,-0.709604990065821,-0.133868544927673,0.128241072050519],[0,0,0,0],[8.999999E+09,8.999999E+09,8.999999E+09,8.999999E+09,8.999999E+09,8.999999E+09]];
	LOCAL CONST Robtarget Tr_meulage_bavure_P435 :=[[2.16424560546875,-116.1051953125,23],[0.678517428853039,-0.709679066641573,-0.137083502758273,0.131064237627695],[0,0,0,0],[8.999999E+09,8.999999E+09,8.999999E+09,8.999999E+09,8.999999E+09,8.999999E+09]];
	LOCAL CONST Robtarget Tr_meulage_bavure_P436 :=[[0.2020263671875,-116.9593828125,23],[0.677211811682237,-0.709720892205289,-0.140438369907851,0.134005528031555],[0,0,0,0],[8.999999E+09,8.999999E+09,8.999999E+09,8.999999E+09,8.999999E+09,8.999999E+09]];
	LOCAL CONST Robtarget Tr_meulage_bavure_P437 :=[[-0.35601806640625,-117.193203125,23],[0.675823463069176,-0.709676363452755,-0.144147807350828,0.137271685199856],[0,0,0,0],[8.999999E+09,8.999999E+09,8.999999E+09,8.999999E+09,8.999999E+09,8.999999E+09]];
	LOCAL CONST Robtarget Tr_meulage_bavure_P438 :=[[-0.874114990234375,-117.41409375,23],[0.674301261294345,-0.709475997301703,-0.148481507171362,0.141120020896152],[0,0,0,0],[8.999999E+09,8.999999E+09,8.999999E+09,8.999999E+09,8.999999E+09,8.999999E+09]];
	LOCAL CONST Robtarget Tr_meulage_bavure_P439 :=[[-3.60552978515625,-118.5310234375,23],[0.672593094841608,-0.709054945041968,-0.153664678067754,0.145762753806495],[0,0,0,0],[8.999999E+09,8.999999E+09,8.999999E+09,8.999999E+09,8.999999E+09,8.999999E+09]];
	LOCAL CONST Robtarget Tr_meulage_bavure_P440 :=[[-4.56396484375,-119.034015625,23],[0.670671869753383,-0.708373756124088,-0.159766446646974,0.151263172259321],[0,0,0,0],[8.999999E+09,8.999999E+09,8.999999E+09,8.999999E+09,8.999999E+09,8.999999E+09]];
	LOCAL CONST Robtarget Tr_meulage_bavure_P441 :=[[-9.8644716796875,-121.5056015625,23],[0.668550552285878,-0.707432095550184,-0.1666570649912,0.157497339381468],[0,0,0,0],[8.999999E+09,8.999999E+09,8.999999E+09,8.999999E+09,8.999999E+09,8.999999E+09]];
	LOCAL CONST Robtarget Tr_meulage_bavure_P442 :=[[-12.75082421875,-123.15509375,23],[0.666279866801151,-0.70627951128807,-0.174031322300158,0.164175180488966],[0,0,0,0],[8.999999E+09,8.999999E+09,8.999999E+09,8.999999E+09,8.999999E+09,8.999999E+09]];
	LOCAL CONST Robtarget Tr_meulage_bavure_P443 :=[[-14.347412109375,-123.9255234375,23],[0.663952333465541,-0.705005890975047,-0.181462537204327,0.170895699675302],[0,0,0,0],[8.999999E+09,8.999999E+09,8.999999E+09,8.999999E+09,8.999999E+09,8.999999E+09]];
	LOCAL CONST Robtarget Tr_meulage_bavure_P444 :=[[-16.77655078125,-125.2828515625,23],[0.661673047938162,-0.703724708703653,-0.188521755625078,0.177256479848327],[0,0,0,0],[8.999999E+09,8.999999E+09,8.999999E+09,8.999999E+09,8.999999E+09,8.999999E+09]];
	LOCAL CONST Robtarget Tr_meulage_bavure_P445 :=[[-19.107208984375,-126.4220390625,23],[0.659538084765806,-0.702530150662635,-0.194894290909275,0.182967531339192],[0,0,0,0],[8.999999E+09,8.999999E+09,8.999999E+09,8.999999E+09,8.999999E+09,8.999999E+09]];
	LOCAL CONST Robtarget Tr_meulage_bavure_P446 :=[[-21.154205078125,-127.7093671875,23],[0.657602809094704,-0.701471611832308,-0.200455537201457,0.187919399928302],[0,0,0,0],[8.999999E+09,8.999999E+09,8.999999E+09,8.999999E+09,8.999999E+09,8.999999E+09]];
	LOCAL CONST Robtarget Tr_meulage_bavure_P447 :=[[-22.304900390625,-128.4650390625,23],[0.655840306614266,-0.700522656859547,-0.205365682379165,0.192266575221712],[0,0,0,0],[8.999999E+09,8.999999E+09,8.999999E+09,8.999999E+09,8.999999E+09,8.999999E+09]];
	LOCAL CONST Robtarget Tr_meulage_bavure_P448 :=[[-24.552947265625,-130.22334375,23],[0.654145961861597,-0.699560880584795,-0.210060515753938,0.19642355932215],[0,0,0,0],[8.999999E+09,8.999999E+09,8.999999E+09,8.999999E+09,8.999999E+09,8.999999E+09]];
	LOCAL CONST Robtarget Tr_meulage_bavure_P449 :=[[-28.655701171875,-132.9463125,23],[0.652337582226603,-0.69838396217471,-0.215198696176503,0.201010052872576],[0,0,0,0],[8.999999E+09,8.999999E+09,8.999999E+09,8.999999E+09,8.999999E+09,8.999999E+09]];
	LOCAL CONST Robtarget Tr_meulage_bavure_P450 :=[[-28.90545703125,-133.129640625,23],[0.650190439844875,-0.696745484395722,-0.221513328512298,0.206712281202403],[0,0,0,0],[8.999999E+09,8.999999E+09,8.999999E+09,8.999999E+09,8.999999E+09,8.999999E+09]];
	LOCAL CONST Robtarget Tr_meulage_bavure_P451 :=[[-29.4898984375,-133.570765625,23],[0.647498337903728,-0.694410523716665,-0.229587988969126,0.214077748223793],[0,0,0,0],[8.999999E+09,8.999999E+09,8.999999E+09,8.999999E+09,8.999999E+09,8.999999E+09]];
	LOCAL CONST Robtarget Tr_meulage_bavure_P452 :=[[-30.609619140625,-134.461046875,23],[0.644118912457013,-0.691218488892223,-0.239676534526797,0.223344993286106],[0,0,0,0],[8.999999E+09,8.999999E+09,8.999999E+09,8.999999E+09,8.999999E+09,8.999999E+09]];
	LOCAL CONST Robtarget Tr_meulage_bavure_P453 :=[[-33.33517578125,-136.900375,23],[0.640043104200405,-0.687150393836731,-0.251542419800352,0.234298041085533],[0,0,0,0],[8.999999E+09,8.999999E+09,8.999999E+09,8.999999E+09,8.999999E+09,8.999999E+09]];
	LOCAL CONST Robtarget Tr_meulage_bavure_P454 :=[[-33.39108203125,-136.9475,23],[0.635417641322253,-0.682358631583968,-0.26450504982436,0.246309150493302],[0,0,0,0],[8.999999E+09,8.999999E+09,8.999999E+09,8.999999E+09,8.999999E+09,8.999999E+09]];
	LOCAL CONST Robtarget Tr_meulage_bavure_P455 :=[[-33.52685546875,-137.093296875,23],[0.630531918642478,-0.677156973206533,-0.277610720405723,0.258496075650325],[0,0,0,0],[8.999999E+09,8.999999E+09,8.999999E+09,8.999999E+09,8.999999E+09,8.999999E+09]];
	LOCAL CONST Robtarget Tr_meulage_bavure_P456 :=[[-38.42575,-142.479109375,23],[0.62575531972449,-0.671937344347846,-0.289901688193979,0.269976843987677],[0,0,0,0],[8.999999E+09,8.999999E+09,8.999999E+09,8.999999E+09,8.999999E+09,8.999999E+09]];
	LOCAL CONST Robtarget Tr_meulage_bavure_P457 :=[[-39.4045703125,-143.64128125,23],[0.621411970199962,-0.667056448985834,-0.300693645922067,0.280118168744381],[0,0,0,0],[8.999999E+09,8.999999E+09,8.999999E+09,8.999999E+09,8.999999E+09,8.999999E+09]];
	LOCAL CONST Robtarget Tr_meulage_bavure_P458 :=[[-42.74878125,-147.818609375,23],[0.617689697854642,-0.662726693933681,-0.309715316577255,0.288667956291351],[0,0,0,0],[8.999999E+09,8.999999E+09,8.999999E+09,8.999999E+09,8.999999E+09,8.999999E+09]];
	LOCAL CONST Robtarget Tr_meulage_bavure_P459 :=[[-42.83279296875,-147.927109375,23],[0.614604779272841,-0.658973631605859,-0.317095356484356,0.295745250239506],[0,0,0,0],[8.999999E+09,8.999999E+09,8.999999E+09,8.999999E+09,8.999999E+09,8.999999E+09]];
	LOCAL CONST Robtarget Tr_meulage_bavure_P460 :=[[-43.38623046875,-148.656640625,23],[0.612022635161427,-0.655666685725701,-0.323246766384133,0.301730043750601],[0,0,0,0],[8.999999E+09,8.999999E+09,8.999999E+09,8.999999E+09,8.999999E+09,8.999999E+09]];
	LOCAL CONST Robtarget Tr_meulage_bavure_P461 :=[[-44.634734375,-150.339296875,23],[0.609740262893897,-0.652605084055821,-0.328670030919456,0.307082117431118],[0,0,0,0],[8.999999E+09,8.999999E+09,8.999999E+09,8.999999E+09,8.999999E+09,8.999999E+09]];
	LOCAL CONST Robtarget Tr_meulage_bavure_P462 :=[[-46.93628125,-153.60746875,23],[0.607563344890476,-0.649603867428823,-0.333793556074992,0.312191382472071],[0,0,0,0],[8.999999E+09,8.999999E+09,8.999999E+09,8.999999E+09,8.999999E+09,8.999999E+09]];
	LOCAL CONST Robtarget Tr_meulage_bavure_P463 :=[[-48.58245703125,-155.930078125,23],[0.605369848735387,-0.646550813629388,-0.338866817883611,0.317283266773882],[0,0,0,0],[8.999999E+09,8.999999E+09,8.999999E+09,8.999999E+09,8.999999E+09,8.999999E+09]];
	LOCAL CONST Robtarget Tr_meulage_bavure_P464 :=[[-48.90243359375,-156.46321875,23],[0.603122647278245,-0.643423455841618,-0.343951272644531,0.322407895156304],[0,0,0,0],[8.999999E+09,8.999999E+09,8.999999E+09,8.999999E+09,8.999999E+09,8.999999E+09]];
	LOCAL CONST Robtarget Tr_meulage_bavure_P465 :=[[-51.0249921875,-159.872796875,23],[0.600835995539512,-0.640260872605313,-0.348998780413848,0.32750873689777],[0,0,0,0],[8.999999E+09,8.999999E+09,8.999999E+09,8.999999E+09,8.999999E+09,8.999999E+09]];
	LOCAL CONST Robtarget Tr_meulage_bavure_P466 :=[[-52.06985546875,-161.604328125,23],[0.598550223472756,-0.637124595623887,-0.353919637033204,0.332491759528108],[0,0,0,0],[8.999999E+09,8.999999E+09,8.999999E+09,8.999999E+09,8.999999E+09,8.999999E+09]];
	LOCAL CONST Robtarget Tr_meulage_bavure_P467 :=[[-52.61065625,-162.602828125,23],[0.59627458773251,-0.634041008491963,-0.358691557022931,0.337326225626448],[0,0,0,0],[8.999999E+09,8.999999E+09,8.999999E+09,8.999999E+09,8.999999E+09,8.999999E+09]];
	LOCAL CONST Robtarget Tr_meulage_bavure_P468 :=[[-53.03857421875,-163.38746875,23],[0.593972681392658,-0.630980712767051,-0.363383511833841,0.342070485722615],[0,0,0,0],[8.999999E+09,8.999999E+09,8.999999E+09,8.999999E+09,8.999999E+09,8.999999E+09]];
	LOCAL CONST Robtarget Tr_meulage_bavure_P469 :=[[-53.2253125,-163.632734375,23],[0.591550661608907,-0.627853664269648,-0.368163697946637,0.346876177515116],[0,0,0,0],[8.999999E+09,8.999999E+09,8.999999E+09,8.999999E+09,8.999999E+09,8.999999E+09]];
	LOCAL CONST Robtarget Tr_meulage_bavure_P470 :=[[-54.46209765625,-165.833984375,23],[0.588874463895087,-0.624523191158417,-0.373262252091175,0.351955878827737],[0,0,0,0],[8.999999E+09,8.999999E+09,8.999999E+09,8.999999E+09,8.999999E+09,8.999999E+09]];
	LOCAL CONST Robtarget Tr_meulage_bavure_P471 :=[[-55.025421875,-166.877359375,23],[0.585819220486955,-0.620856280698047,-0.378878667245573,0.357497237936271],[0,0,0,0],[8.999999E+09,8.999999E+09,8.999999E+09,8.999999E+09,8.999999E+09,8.999999E+09]];
	LOCAL CONST Robtarget Tr_meulage_bavure_P472 :=[[-55.4491875,-167.804359375,23],[0.58230911800569,-0.616771317411469,-0.385110302262946,0.36359220040713],[0,0,0,0],[8.999999E+09,8.999999E+09,8.999999E+09,8.999999E+09,8.999999E+09,8.999999E+09]];
	LOCAL CONST Robtarget Tr_meulage_bavure_P473 :=[[-57.186125,-171.569515625,23],[0.578376752808909,-0.612300979151903,-0.391862128643576,0.370151205421201],[0,0,0,0],[8.999999E+09,8.999999E+09,8.999999E+09,8.999999E+09,8.999999E+09,8.999999E+09]];
	LOCAL CONST Robtarget Tr_meulage_bavure_P474 :=[[-58.07678125,-173.466140625,23],[0.574202680396625,-0.607625333075722,-0.398809886070948,0.376873203082982],[0,0,0,0],[8.999999E+09,8.999999E+09,8.999999E+09,8.999999E+09,8.999999E+09,8.999999E+09]];
	LOCAL CONST Robtarget Tr_meulage_bavure_P475 :=[[-58.51434375,-174.5696875,23],[0.570093809639072,-0.603056034680678,-0.4054607927701,0.383298855689223],[0,0,0,0],[8.999999E+09,8.999999E+09,8.999999E+09,8.999999E+09,8.999999E+09,8.999999E+09]];
	LOCAL CONST Robtarget Tr_meulage_bavure_P476 :=[[-60.36853125,-179.709046875,23],[0.566439217206491,-0.598997920097138,-0.411237895412486,0.388884942247075],[0,0,0,0],[8.999999E+09,8.999999E+09,8.999999E+09,8.999999E+09,8.999999E+09,8.999999E+09]];
	LOCAL CONST Robtarget Tr_meulage_bavure_P477 :=[[-61.01123046875,-181.3869375,23],[0.563599857332851,-0.595825735452697,-0.415650008601314,0.393169129175181],[0,0,0,0],[8.999999E+09,8.999999E+09,8.999999E+09,8.999999E+09,8.999999E+09,8.999999E+09]];
	LOCAL CONST Robtarget Tr_meulage_bavure_P478 :=[[-61.25525,-182.19803125,23],[0.561802271074709,-0.593760614964307,-0.418429538840201,0.395908147628315],[0,0,0,0],[8.999999E+09,8.999999E+09,8.999999E+09,8.999999E+09,8.999999E+09,8.999999E+09]];
	LOCAL CONST Robtarget Tr_meulage_bavure_P479 :=[[-61.6721171875,-183.65096875,23],[0.561001629658851,-0.592746351096124,-0.419696774248578,0.397219778545432],[0,0,0,0],[8.999999E+09,8.999999E+09,8.999999E+09,8.999999E+09,8.999999E+09,8.999999E+09]];
	LOCAL CONST Robtarget Tr_meulage_bavure_P480 :=[[-62.20779296875,-185.31396875,23],[0.560795967876218,-0.592349764131507,-0.420076800028189,0.397699788062805],[0,0,0,0],[8.999999E+09,8.999999E+09,8.999999E+09,8.999999E+09,8.999999E+09,8.999999E+09]];
	LOCAL CONST Robtarget Tr_meulage_bavure_P481 :=[[-62.853453125,-187.8425,23],[0.560487467395075,-0.59183144645005,-0.420614090950561,0.39833795247218],[0,0,0,0],[8.999999E+09,8.999999E+09,8.999999E+09,8.999999E+09,8.999999E+09,8.999999E+09]];
	LOCAL CONST Robtarget Tr_meulage_bavure_P482 :=[[-63.188875,-189.049921875,23],[0.559251310085681,-0.590318665684458,-0.422527332441281,0.400290517564462],[0,0,0,0],[8.999999E+09,8.999999E+09,8.999999E+09,8.999999E+09,8.999999E+09,8.999999E+09]];
	LOCAL CONST Robtarget Tr_meulage_bavure_P483 :=[[-63.375671875,-189.785640625,23],[0.556418329778567,-0.587104033860667,-0.426759787208525,0.404454669564709],[0,0,0,0],[8.999999E+09,8.999999E+09,8.999999E+09,8.999999E+09,8.999999E+09,8.999999E+09]];
	LOCAL CONST Robtarget Tr_meulage_bavure_P484 :=[[-63.64144921875,-190.991640625,23],[0.551716955328234,-0.581908891844406,-0.433585324452152,0.411089052658279],[0,0,0,0],[8.999999E+09,8.999999E+09,8.999999E+09,8.999999E+09,8.999999E+09,8.999999E+09]];
	LOCAL CONST Robtarget Tr_meulage_bavure_P485 :=[[-64.199921875,-193.55175,23],[0.545403815288625,-0.575013063516636,-0.442457371647882,0.419673836840317],[0,0,0,0],[8.999999E+09,8.999999E+09,8.999999E+09,8.999999E+09,8.999999E+09,8.999999E+09]];
	LOCAL CONST Robtarget Tr_meulage_bavure_P486 :=[[-64.85885546875,-197.687890625,23],[0.538169851316207,-0.567154569131266,-0.452261528733606,0.429148477191009],[0,0,0,0],[8.999999E+09,8.999999E+09,8.999999E+09,8.999999E+09,8.999999E+09,8.999999E+09]];
	LOCAL CONST Robtarget Tr_meulage_bavure_P487 :=[[-64.9612421875,-198.337671875,23],[0.530875345552407,-0.55925576444528,-0.461789245240804,0.438354936551725],[0,0,0,0],[8.999999E+09,8.999999E+09,8.999999E+09,8.999999E+09,8.999999E+09,8.999999E+09]];
	LOCAL CONST Robtarget Tr_meulage_bavure_P488 :=[[-65.13421484375,-200.074640625,23],[0.524236559480971,-0.552079561165831,-0.470169814028609,0.446457762641441],[0,0,0,0],[8.999999E+09,8.999999E+09,8.999999E+09,8.999999E+09,8.999999E+09,8.999999E+09]];
	LOCAL CONST Robtarget Tr_meulage_bavure_P489 :=[[-65.43667578125,-202.296875,23],[0.518686994011296,-0.546092871717492,-0.476973871723315,0.453036757224112],[0,0,0,0],[8.999999E+09,8.999999E+09,8.999999E+09,8.999999E+09,8.999999E+09,8.999999E+09]];
	LOCAL CONST Robtarget Tr_meulage_bavure_P490 :=[[-65.51962109375,-203.27371875,23],[0.514492371399699,-0.541584091869836,-0.481998943321615,0.45788785727718],[0,0,0,0],[8.999999E+09,8.999999E+09,8.999999E+09,8.999999E+09,8.999999E+09,8.999999E+09]];
	LOCAL CONST Robtarget Tr_meulage_bavure_P491 :=[[-65.660828125,-204.464453125,23],[0.511935512769435,-0.538861064211317,-0.485011219497922,0.460776411292593],[0,0,0,0],[8.999999E+09,8.999999E+09,8.999999E+09,8.999999E+09,8.999999E+09,8.999999E+09]];
	LOCAL CONST Robtarget Tr_meulage_bavure_P492 :=[[-65.7692578125,-208.40615625,23],[0.511546789799372,-0.53849022574215,-0.485459477214173,0.461169442406006],[0,0,0,0],[8.999999E+09,8.999999E+09,8.999999E+09,8.999999E+09,8.999999E+09,8.999999E+09]];
	LOCAL CONST Robtarget Tr_meulage_bavure_P493 :=[[-65.809078125,-209.24296875,23],[0.51410710296833,-0.54130002139387,-0.482433963452917,0.458198258861397],[0,0,0,0],[8.999999E+09,8.999999E+09,8.999999E+09,8.999999E+09,8.999999E+09,8.999999E+09]];
	LOCAL CONST Robtarget Tr_meulage_bavure_P494 :=[[-65.8337421875,-209.985875,23],[0.520420879209584,-0.548143807941173,-0.474831544508943,0.450816457815955],[0,0,0,0],[8.999999E+09,8.999999E+09,8.999999E+09,8.999999E+09,8.999999E+09,8.999999E+09]];
	LOCAL CONST Robtarget Tr_meulage_bavure_P495 :=[[-65.6136796875,-214.05571875,23],[0.530903751891648,-0.559467348146617,-0.461708281492133,0.438135772776824],[0,0,0,0],[8.999999E+09,8.999999E+09,8.999999E+09,8.999999E+09,8.999999E+09,8.999999E+09]];
	LOCAL CONST Robtarget Tr_meulage_bavure_P496 :=[[-65.478453125,-215.351453125,23],[0.545155302506434,-0.574857600784445,-0.44276371195308,0.419886568428903],[0,0,0,0],[8.999999E+09,8.999999E+09,8.999999E+09,8.999999E+09,8.999999E+09,8.999999E+09]];
	LOCAL CONST Robtarget Tr_meulage_bavure_P497 :=[[-65.49206640625,-216.463,23],[0.56182588988593,-0.592897593598313,-0.418761655858971,0.396815811859185],[0,0,0,0],[8.999999E+09,8.999999E+09,8.999999E+09,8.999999E+09,8.999999E+09,8.999999E+09]];
	LOCAL CONST Robtarget Tr_meulage_bavure_P498 :=[[-65.5283515625,-217.137421875,23],[0.578970879669977,-0.611535084853853,-0.39160903696482,0.370755880134692],[0,0,0,0],[8.999999E+09,8.999999E+09,8.999999E+09,8.999999E+09,8.999999E+09,8.999999E+09]];
	LOCAL CONST Robtarget Tr_meulage_bavure_P499 :=[[-65.953125,-219.276375,23],[0.59491132776535,-0.628990647907625,-0.363584934132002,0.343885551620655],[0,0,0,0],[8.999999E+09,8.999999E+09,8.999999E+09,8.999999E+09,8.999999E+09,8.999999E+09]];
	LOCAL CONST Robtarget Tr_meulage_bavure_P500 :=[[-66.02459375,-219.75290625,23],[0.608972643939836,-0.644531003317206,-0.336041892895242,0.317502678595352],[0,0,0,0],[8.999999E+09,8.999999E+09,8.999999E+09,8.999999E+09,8.999999E+09,8.999999E+09]];
	LOCAL CONST Robtarget Tr_meulage_bavure_P501 :=[[-66.1534140625,-219.90875,23],[0.621505009452641,-0.658505117118502,-0.308630820641154,0.291289461711865],[0,0,0,0],[8.999999E+09,8.999999E+09,8.999999E+09,8.999999E+09,8.999999E+09,8.999999E+09]];
	LOCAL CONST Robtarget Tr_meulage_bavure_P502 :=[[-67.90503125,-221.502703125,23],[0.633313388925439,-0.671747452401822,-0.279606610884595,0.263608904912312],[0,0,0,0],[8.999999E+09,8.999999E+09,8.999999E+09,8.999999E+09,8.999999E+09,8.999999E+09]];
	LOCAL CONST Robtarget Tr_meulage_bavure_P503 :=[[-68.539,-221.773828125,23],[0.644933607098693,-0.684801550877158,-0.246985377898685,0.232606322904497],[0,0,0,0],[8.999999E+09,8.999999E+09,8.999999E+09,8.999999E+09,8.999999E+09,8.999999E+09]];
	LOCAL CONST Robtarget Tr_meulage_bavure_P504 :=[[-70.7229296875,-222.56971875,23],[0.656099990520838,-0.697363578337009,-0.210102666257281,0.197670715279581],[0,0,0,0],[8.999999E+09,8.999999E+09,8.999999E+09,8.999999E+09,8.999999E+09,8.999999E+09]];
	LOCAL CONST Robtarget Tr_meulage_bavure_P505 :=[[-71.4143984375,-222.65475,23],[0.665838821081493,-0.708375341972006,-0.1706695301687,0.160421166617273],[0,0,0,0],[8.999999E+09,8.999999E+09,8.999999E+09,8.999999E+09,8.999999E+09,8.999999E+09]];
	LOCAL CONST Robtarget Tr_meulage_bavure_P506 :=[[-73.9191875,-223.039578125,23],[0.673182689245091,-0.716783138923678,-0.132510749147552,0.12445039178653],[0,0,0,0],[8.999999E+09,8.999999E+09,8.999999E+09,8.999999E+09,8.999999E+09,8.999999E+09]];
	LOCAL CONST Robtarget Tr_meulage_bavure_P507 :=[[-75.83334375,-223.166078125,23],[0.677899805297806,-0.722321494560677,-0.0997222349547708,0.0935894669738676],[0,0,0,0],[8.999999E+09,8.999999E+09,8.999999E+09,8.999999E+09,8.999999E+09,8.999999E+09]];
	LOCAL CONST Robtarget Tr_meulage_bavure_P508 :=[[-77.405640625,-223.295171875,23],[0.680519173132546,-0.725525032953498,-0.074763066815951,0.0701253548803537],[0,0,0,0],[8.999999E+09,8.999999E+09,8.999999E+09,8.999999E+09,8.999999E+09,8.999999E+09]];
	LOCAL CONST Robtarget Tr_meulage_bavure_P509 :=[[-79.190640625,-223.471953125,23],[0.681799034707915,-0.727192620008582,-0.0580909674157705,0.0544647517309153],[0,0,0,0],[8.999999E+09,8.999999E+09,8.999999E+09,8.999999E+09,8.999999E+09,8.999999E+09]];
	LOCAL CONST Robtarget Tr_meulage_bavure_P510 :=[[-85.158078125,-224.142265625,23],[0.682344059453636,-0.727959051338062,-0.0488459151636144,0.0457851578041446],[0,0,0,0],[8.999999E+09,8.999999E+09,8.999999E+09,8.999999E+09,8.999999E+09,8.999999E+09]];
	LOCAL CONST Robtarget Tr_meulage_bavure_P511 :=[[-86.355375,-224.2940625,23],[0.682491944699804,-0.728178301528877,-0.0459206313267657,0.0430395425272147],[0,0,0,0],[8.999999E+09,8.999999E+09,8.999999E+09,8.999999E+09,8.999999E+09,8.999999E+09]];
	LOCAL CONST Robtarget Tr_meulage_bavure_degg1 :=[[-85.1017565609581,-234.194050942676,23.6470468639786],[0.682491944699804,-0.728178301528877,-0.0459206313267657,0.0430395425272147],[0,0,0,0],[8.999999E+09,8.999999E+09,8.999999E+09,8.999999E+09,8.999999E+09,8.999999E+09]];
	LOCAL CONST Robtarget Tr_meulage_bavure_degg2 :=[[-61.2830062191623,-422.293831353511,35.9409372795713],[0.682491944699804,-0.728178301528877,-0.0459206313267657,0.0430395425272147],[0,0,0,0],[8.999999E+09,8.999999E+09,8.999999E+09,8.999999E+09,8.999999E+09,8.999999E+09]];
	LOCAL PROC Tr_pick()
		!!Programme Tr_pick - 24/03/2023 10:23:34;
		 CONST Robtarget Ppick :=[[1.94688526622454,5.56235420550051,45.2471422487626],[-0.0030677707191134,-0.883414684365503,-0.468327257416204,-0.0154487601842293],[0,0,0,0],[8.999999E+09,8.999999E+09,8.999999E+09,8.999999E+09,8.999999E+09,8.999999E+09]];
		 VAR Pose Ref :=[[0,0,0],[1,0,0,0]];
		LocalisationPieceTable 90 \model:=0;
		MoveJ Reltool(Ppick,0,0,-200),V1000,Z0,Tool_Prehenseur \Wobj:=Wobj_vision;
		MoveL Reltool(Ppick,0,0,-100),V500,Z0,Tool_Prehenseur \Wobj:=Wobj_vision;
		MoveL Reltool(Ppick,0,0,-10),V200,Z0,Tool_Prehenseur \Wobj:=Wobj_vision;
		MoveL Ppick,V100,Fine,Tool_Prehenseur \Wobj:=Wobj_vision;
		Gripper_Close;
		MoveL Reltool(Ppick,0,0,-200),V500,Z0,Tool_Prehenseur \Wobj:=Wobj_vision;
		LocalisationPiecePrehenseur 90 \model:=0,Ref;
	ENDPROC
	LOCAL PROC Tr_Cut()
		!!Programme Tr_Cut - 24/03/2023 10:23:34;
		confJ \off;
		confL \off;
		Tool := ToolOffset(Tool_M2_D490_S180);
		MoveAbsJ [[0,-40,40,0,90,0],[8.999999E+09,8.999999E+09,8.999999E+09,8.999999E+09,8.999999E+09,8.999999E+09]] ,V1000,Z0,Tool_M2_D490_S180 \Wobj:=Wobj_Part_0;
		Movej Reltool(Coupe_0,-200,0,-43.35395703125),V1000,Z0,Tool_M2_D490_S180 \Wobj:=Wobj_Part_0;
		MoveL Reltool(Coupe_0,0,0,-43.35395703125),V500,Z0,Tool_M2_D490_S180 \Wobj:=Wobj_Part_0;
		MoveL Reltool(Coupe_0,0,0,-33.35395703125),vitesse_Tronconnage,Z0,Tool_M2_D490_S180 \Wobj:=Wobj_Part_0;
		MoveL Coupe_0,vitesse_Tronconnage,Fine,Tool_M2_D490_S180 \Wobj:=Wobj_Part_0;
		MoveL Reltool(Coupe_0,0,0,33.35395703125),vitesse_Tronconnage,Z0,Tool_M2_D490_S180 \Wobj:=Wobj_Part_0;
		MoveL Reltool(Coupe_0,-200,0,33.35395703125),V500,Z0,Tool_M2_D490_S180 \Wobj:=Wobj_Part_0;
		MoveAbsJ [[0,-40,40,0,90,0],[8.999999E+09,8.999999E+09,8.999999E+09,8.999999E+09,8.999999E+09,8.999999E+09]] ,V1000,Z0,Tool_M2_D490_S180 \Wobj:=Wobj_Part_0;
		Movej Reltool(Coupe_1,-200,0,-35.65858203125),V1000,Z0,Tool_M2_D490_S180 \Wobj:=Wobj_Part_0;
		MoveL Reltool(Coupe_1,0,0,-35.65858203125),V500,Z0,Tool_M2_D490_S180 \Wobj:=Wobj_Part_0;
		MoveL Reltool(Coupe_1,0,0,-25.65858203125),vitesse_Tronconnage,Z0,Tool_M2_D490_S180 \Wobj:=Wobj_Part_0;
		MoveL Coupe_1,vitesse_Tronconnage,Fine,Tool_M2_D490_S180 \Wobj:=Wobj_Part_0;
		MoveL Reltool(Coupe_1,0,0,25.65858203125),vitesse_Tronconnage,Z0,Tool_M2_D490_S180 \Wobj:=Wobj_Part_0;
		MoveL Reltool(Coupe_1,-200,0,25.65858203125),V500,Z0,Tool_M2_D490_S180 \Wobj:=Wobj_Part_0;
	ENDPROC
	LOCAL PROC Tr_meulage_motif_1()
		!!Programme Tr_meulage_motif_1 - 24/03/2023 10:23:34;
		 CONST Speeddata vitesse_Meulage :=[50, 500, 0, 0];
		confJ \off;
		confL \off;
		Tool := ToolOffset(Tool_M1_D500_S0);
		MoveAbsJ [[0,-40,40,0,90,0],[8.999999E+09,8.999999E+09,8.999999E+09,8.999999E+09,8.999999E+09,8.999999E+09]] ,V1000,Z0,Tool_M1_D500_S0 \Wobj:=Wobj_Part_0;
		MoveJ Tr_meulage_motif_1_App1,V2000,Z100,Tool,\Wobj:=Wobj_Part_0;
		MoveJ Tr_meulage_motif_1_App2,V500,Z0,Tool,\Wobj:=Wobj_Part_0;
		MoveL Tr_meulage_motif_1_P0,[12.5,500,0,0],z0,Tool \wobj:=Wobj_Part_0;
		MoveL Tr_meulage_motif_1_P1,[12.5,500,0,0],z0,Tool \wobj:=Wobj_Part_0;
		MoveL Tr_meulage_motif_1_P2,[12.5,500,0,0],z0,Tool \wobj:=Wobj_Part_0;
		MoveL Tr_meulage_motif_1_P3,[12.5,500,0,0],z0,Tool \wobj:=Wobj_Part_0;
		MoveL Tr_meulage_motif_1_P4,[12.5,500,0,0],z0,Tool \wobj:=Wobj_Part_0;
		MoveL Tr_meulage_motif_1_P5,[12.5,500,0,0],z0,Tool \wobj:=Wobj_Part_0;
		MoveL Tr_meulage_motif_1_P6,[12.5,500,0,0],z0,Tool \wobj:=Wobj_Part_0;
		MoveL Tr_meulage_motif_1_P7,[12.5,500,0,0],z0,Tool \wobj:=Wobj_Part_0;
		MoveL Tr_meulage_motif_1_P8,[12.5,500,0,0],z0,Tool \wobj:=Wobj_Part_0;
		MoveL Tr_meulage_motif_1_P9,[12.5,500,0,0],z0,Tool \wobj:=Wobj_Part_0;
		MoveL Tr_meulage_motif_1_P10,[12.5,500,0,0],z0,Tool \wobj:=Wobj_Part_0;
		MoveL Tr_meulage_motif_1_P11,[12.5,500,0,0],z0,Tool \wobj:=Wobj_Part_0;
		MoveL Tr_meulage_motif_1_P12,[12.5,500,0,0],z0,Tool \wobj:=Wobj_Part_0;
		MoveL Tr_meulage_motif_1_P13,[12.5,500,0,0],z0,Tool \wobj:=Wobj_Part_0;
		MoveL Tr_meulage_motif_1_P14,[12.5,500,0,0],z0,Tool \wobj:=Wobj_Part_0;
		MoveL Tr_meulage_motif_1_P15,[12.5,500,0,0],z0,Tool \wobj:=Wobj_Part_0;
		MoveL Tr_meulage_motif_1_P16,[12.5,500,0,0],z0,Tool \wobj:=Wobj_Part_0;
		MoveL Tr_meulage_motif_1_P17,[12.5,500,0,0],z0,Tool \wobj:=Wobj_Part_0;
		MoveL Tr_meulage_motif_1_P18,[12.5,500,0,0],z0,Tool \wobj:=Wobj_Part_0;
		MoveL Tr_meulage_motif_1_P19,[12.5,500,0,0],z0,Tool \wobj:=Wobj_Part_0;
		MoveL Tr_meulage_motif_1_P20,[12.5,500,0,0],z0,Tool \wobj:=Wobj_Part_0;
		MoveL Tr_meulage_motif_1_P21,[12.5,500,0,0],z0,Tool \wobj:=Wobj_Part_0;
		MoveL Tr_meulage_motif_1_P22,[12.5,500,0,0],z0,Tool \wobj:=Wobj_Part_0;
		MoveL Tr_meulage_motif_1_P23,[12.5,500,0,0],z0,Tool \wobj:=Wobj_Part_0;
		MoveL Tr_meulage_motif_1_P24,[12.5,500,0,0],z0,Tool \wobj:=Wobj_Part_0;
		MoveL Tr_meulage_motif_1_P25,[12.5,500,0,0],z0,Tool \wobj:=Wobj_Part_0;
		MoveL Tr_meulage_motif_1_P26,[12.5,500,0,0],z0,Tool \wobj:=Wobj_Part_0;
		MoveL Tr_meulage_motif_1_P27,[12.5,500,0,0],z0,Tool \wobj:=Wobj_Part_0;
		MoveL Tr_meulage_motif_1_P28,[12.5,500,0,0],z0,Tool \wobj:=Wobj_Part_0;
		MoveL Tr_meulage_motif_1_P29,[12.5,500,0,0],z0,Tool \wobj:=Wobj_Part_0;
		MoveL Tr_meulage_motif_1_P30,[12.5,500,0,0],z0,Tool \wobj:=Wobj_Part_0;
		MoveL Tr_meulage_motif_1_P31,[12.5,500,0,0],z0,Tool \wobj:=Wobj_Part_0;
		MoveL Tr_meulage_motif_1_P32,[12.5,500,0,0],z0,Tool \wobj:=Wobj_Part_0;
		MoveL Tr_meulage_motif_1_P33,[12.5,500,0,0],z0,Tool \wobj:=Wobj_Part_0;
		MoveL Tr_meulage_motif_1_P34,[12.5,500,0,0],z0,Tool \wobj:=Wobj_Part_0;
